//     PlcTask Outputs/GVL_iXlinker.Device_2_EtherCAT.Term_9_EK1100.Term_10_EK1122.Term_23_EK1100.Term_32_EL2258.MTO_Outputs_10x_Channel_6.Output_event_time[1] <-> MTO Outputs 10x Channel 6/Output event time 2
//     PlcTask Outputs/GVL_iXlinker.Device_2_EtherCAT.Term_9_EK1100.Term_10_EK1122.Term_23_EK1100.Term_32_EL2258.MTO_Outputs_10x_Channel_6.Output_event_time[2] <-> MTO Outputs 10x Channel 6/Output event time 3
//     PlcTask Outputs/GVL_iXlinker.Device_2_EtherCAT.Term_9_EK1100.Term_10_EK1122.Term_23_EK1100.Term_32_EL2258.MTO_Outputs_10x_Channel_6.Output_event_time[3] <-> MTO Outputs 10x Channel 6/Output event time 4
//     PlcTask Outputs/GVL_iXlinker.Device_2_EtherCAT.Term_9_EK1100.Term_10_EK1122.Term_23_EK1100.Term_32_EL2258.MTO_Outputs_10x_Channel_6.Output_event_time[4] <-> MTO Outputs 10x Channel 6/Output event time 5
//     PlcTask Outputs/GVL_iXlinker.Device_2_EtherCAT.Term_9_EK1100.Term_10_EK1122.Term_23_EK1100.Term_32_EL2258.MTO_Outputs_10x_Channel_6.Output_event_time[5] <-> MTO Outputs 10x Channel 6/Output event time 6
//     PlcTask Outputs/GVL_iXlinker.Device_2_EtherCAT.Term_9_EK1100.Term_10_EK1122.Term_23_EK1100.Term_32_EL2258.MTO_Outputs_10x_Channel_6.Output_event_time[6] <-> MTO Outputs 10x Channel 6/Output event time 7
//     PlcTask Outputs/GVL_iXlinker.Device_2_EtherCAT.Term_9_EK1100.Term_10_EK1122.Term_23_EK1100.Term_32_EL2258.MTO_Outputs_10x_Channel_6.Output_event_time[7] <-> MTO Outputs 10x Channel 6/Output event time 8
//     PlcTask Outputs/GVL_iXlinker.Device_2_EtherCAT.Term_9_EK1100.Term_10_EK1122.Term_23_EK1100.Term_32_EL2258.MTO_Outputs_10x_Channel_6.Output_event_time[8] <-> MTO Outputs 10x Channel 6/Output event time 9
//     PlcTask Outputs/GVL_iXlinker.Device_2_EtherCAT.Term_9_EK1100.Term_10_EK1122.Term_23_EK1100.Term_32_EL2258.MTO_Outputs_10x_Channel_6.Output_event_time[9] <-> MTO Outputs 10x Channel 6/Output event time 10
//     PlcTask Outputs/GVL_iXlinker.Device_2_EtherCAT.Term_9_EK1100.Term_10_EK1122.Term_23_EK1100.Term_32_EL2258.MTO_Outputs_10x_Channel_7.Output_event_time[0] <-> MTO Outputs 10x Channel 7/Output event time 1
//     PlcTask Outputs/GVL_iXlinker.Device_2_EtherCAT.Term_9_EK1100.Term_10_EK1122.Term_23_EK1100.Term_32_EL2258.MTO_Outputs_10x_Channel_7.Output_event_time[1] <-> MTO Outputs 10x Channel 7/Output event time 2
//     PlcTask Outputs/GVL_iXlinker.Device_2_EtherCAT.Term_9_EK1100.Term_10_EK1122.Term_23_EK1100.Term_32_EL2258.MTO_Outputs_10x_Channel_7.Output_event_time[2] <-> MTO Outputs 10x Channel 7/Output event time 3
//     PlcTask Outputs/GVL_iXlinker.Device_2_EtherCAT.Term_9_EK1100.Term_10_EK1122.Term_23_EK1100.Term_32_EL2258.MTO_Outputs_10x_Channel_7.Output_event_time[3] <-> MTO Outputs 10x Channel 7/Output event time 4
//     PlcTask Outputs/GVL_iXlinker.Device_2_EtherCAT.Term_9_EK1100.Term_10_EK1122.Term_23_EK1100.Term_32_EL2258.MTO_Outputs_10x_Channel_7.Output_event_time[4] <-> MTO Outputs 10x Channel 7/Output event time 5
//     PlcTask Outputs/GVL_iXlinker.Device_2_EtherCAT.Term_9_EK1100.Term_10_EK1122.Term_23_EK1100.Term_32_EL2258.MTO_Outputs_10x_Channel_7.Output_event_time[5] <-> MTO Outputs 10x Channel 7/Output event time 6
//     PlcTask Outputs/GVL_iXlinker.Device_2_EtherCAT.Term_9_EK1100.Term_10_EK1122.Term_23_EK1100.Term_32_EL2258.MTO_Outputs_10x_Channel_7.Output_event_time[6] <-> MTO Outputs 10x Channel 7/Output event time 7
//     PlcTask Outputs/GVL_iXlinker.Device_2_EtherCAT.Term_9_EK1100.Term_10_EK1122.Term_23_EK1100.Term_32_EL2258.MTO_Outputs_10x_Channel_7.Output_event_time[7] <-> MTO Outputs 10x Channel 7/Output event time 8
//     PlcTask Outputs/GVL_iXlinker.Device_2_EtherCAT.Term_9_EK1100.Term_10_EK1122.Term_23_EK1100.Term_32_EL2258.MTO_Outputs_10x_Channel_7.Output_event_time[8] <-> MTO Outputs 10x Channel 7/Output event time 9
//     PlcTask Outputs/GVL_iXlinker.Device_2_EtherCAT.Term_9_EK1100.Term_10_EK1122.Term_23_EK1100.Term_32_EL2258.MTO_Outputs_10x_Channel_7.Output_event_time[9] <-> MTO Outputs 10x Channel 7/Output event time 10
//     PlcTask Outputs/GVL_iXlinker.Device_2_EtherCAT.Term_9_EK1100.Term_10_EK1122.Term_23_EK1100.Term_32_EL2258.MTO_Outputs_10x_Channel_8.Output_event_time[0] <-> MTO Outputs 10x Channel 8/Output event time 1
//     PlcTask Outputs/GVL_iXlinker.Device_2_EtherCAT.Term_9_EK1100.Term_10_EK1122.Term_23_EK1100.Term_32_EL2258.MTO_Outputs_10x_Channel_8.Output_event_time[1] <-> MTO Outputs 10x Channel 8/Output event time 2
//     PlcTask Outputs/GVL_iXlinker.Device_2_EtherCAT.Term_9_EK1100.Term_10_EK1122.Term_23_EK1100.Term_32_EL2258.MTO_Outputs_10x_Channel_8.Output_event_time[2] <-> MTO Outputs 10x Channel 8/Output event time 3
//     PlcTask Outputs/GVL_iXlinker.Device_2_EtherCAT.Term_9_EK1100.Term_10_EK1122.Term_23_EK1100.Term_32_EL2258.MTO_Outputs_10x_Channel_8.Output_event_time[3] <-> MTO Outputs 10x Channel 8/Output event time 4
//     PlcTask Outputs/GVL_iXlinker.Device_2_EtherCAT.Term_9_EK1100.Term_10_EK1122.Term_23_EK1100.Term_32_EL2258.MTO_Outputs_10x_Channel_8.Output_event_time[4] <-> MTO Outputs 10x Channel 8/Output event time 5
//     PlcTask Outputs/GVL_iXlinker.Device_2_EtherCAT.Term_9_EK1100.Term_10_EK1122.Term_23_EK1100.Term_32_EL2258.MTO_Outputs_10x_Channel_8.Output_event_time[5] <-> MTO Outputs 10x Channel 8/Output event time 6
//     PlcTask Outputs/GVL_iXlinker.Device_2_EtherCAT.Term_9_EK1100.Term_10_EK1122.Term_23_EK1100.Term_32_EL2258.MTO_Outputs_10x_Channel_8.Output_event_time[6] <-> MTO Outputs 10x Channel 8/Output event time 7
//     PlcTask Outputs/GVL_iXlinker.Device_2_EtherCAT.Term_9_EK1100.Term_10_EK1122.Term_23_EK1100.Term_32_EL2258.MTO_Outputs_10x_Channel_8.Output_event_time[7] <-> MTO Outputs 10x Channel 8/Output event time 8
//     PlcTask Outputs/GVL_iXlinker.Device_2_EtherCAT.Term_9_EK1100.Term_10_EK1122.Term_23_EK1100.Term_32_EL2258.MTO_Outputs_10x_Channel_8.Output_event_time[8] <-> MTO Outputs 10x Channel 8/Output event time 9
//     PlcTask Outputs/GVL_iXlinker.Device_2_EtherCAT.Term_9_EK1100.Term_10_EK1122.Term_23_EK1100.Term_32_EL2258.MTO_Outputs_10x_Channel_8.Output_event_time[9] <-> MTO Outputs 10x Channel 8/Output event time 10
//     PlcTask Outputs/GVL_iXlinker.Device_2_EtherCAT.Term_9_EK1100.Term_10_EK1122.Term_23_EK1100.Term_32_EL2258.MTO_Outputs_10x_Channel_1.Outputs/Output_event_state_1 <-> MTO Outputs 10x Channel 1/Outputs/Output event state 1
//     PlcTask Outputs/GVL_iXlinker.Device_2_EtherCAT.Term_9_EK1100.Term_10_EK1122.Term_23_EK1100.Term_32_EL2258.MTO_Outputs_10x_Channel_1.Outputs/Output_event_state_10 <-> MTO Outputs 10x Channel 1/Outputs/Output event state 10
//     PlcTask Outputs/GVL_iXlinker.Device_2_EtherCAT.Term_9_EK1100.Term_10_EK1122.Term_23_EK1100.Term_32_EL2258.MTO_Outputs_10x_Channel_1.Outputs/Output_event_state_2 <-> MTO Outputs 10x Channel 1/Outputs/Output event state 2
//     PlcTask Outputs/GVL_iXlinker.Device_2_EtherCAT.Term_9_EK1100.Term_10_EK1122.Term_23_EK1100.Term_32_EL2258.MTO_Outputs_10x_Channel_1.Outputs/Output_event_state_3 <-> MTO Outputs 10x Channel 1/Outputs/Output event state 3
//     PlcTask Outputs/GVL_iXlinker.Device_2_EtherCAT.Term_9_EK1100.Term_10_EK1122.Term_23_EK1100.Term_32_EL2258.MTO_Outputs_10x_Channel_1.Outputs/Output_event_state_4 <-> MTO Outputs 10x Channel 1/Outputs/Output event state 4
//     PlcTask Outputs/GVL_iXlinker.Device_2_EtherCAT.Term_9_EK1100.Term_10_EK1122.Term_23_EK1100.Term_32_EL2258.MTO_Outputs_10x_Channel_1.Outputs/Output_event_state_5 <-> MTO Outputs 10x Channel 1/Outputs/Output event state 5
//     PlcTask Outputs/GVL_iXlinker.Device_2_EtherCAT.Term_9_EK1100.Term_10_EK1122.Term_23_EK1100.Term_32_EL2258.MTO_Outputs_10x_Channel_1.Outputs/Output_event_state_6 <-> MTO Outputs 10x Channel 1/Outputs/Output event state 6
//     PlcTask Outputs/GVL_iXlinker.Device_2_EtherCAT.Term_9_EK1100.Term_10_EK1122.Term_23_EK1100.Term_32_EL2258.MTO_Outputs_10x_Channel_1.Outputs/Output_event_state_7 <-> MTO Outputs 10x Channel 1/Outputs/Output event state 7
//     PlcTask Outputs/GVL_iXlinker.Device_2_EtherCAT.Term_9_EK1100.Term_10_EK1122.Term_23_EK1100.Term_32_EL2258.MTO_Outputs_10x_Channel_1.Outputs/Output_event_state_8 <-> MTO Outputs 10x Channel 1/Outputs/Output event state 8
//     PlcTask Outputs/GVL_iXlinker.Device_2_EtherCAT.Term_9_EK1100.Term_10_EK1122.Term_23_EK1100.Term_32_EL2258.MTO_Outputs_10x_Channel_1.Outputs/Output_event_state_9 <-> MTO Outputs 10x Channel 1/Outputs/Output event state 9
//     PlcTask Outputs/GVL_iXlinker.Device_2_EtherCAT.Term_9_EK1100.Term_10_EK1122.Term_23_EK1100.Term_32_EL2258.MTO_Outputs_10x_Channel_2.Outputs/Output_event_state_1 <-> MTO Outputs 10x Channel 2/Outputs/Output event state 1
//     PlcTask Outputs/GVL_iXlinker.Device_2_EtherCAT.Term_9_EK1100.Term_10_EK1122.Term_23_EK1100.Term_32_EL2258.MTO_Outputs_10x_Channel_2.Outputs/Output_event_state_10 <-> MTO Outputs 10x Channel 2/Outputs/Output event state 10
//     PlcTask Outputs/GVL_iXlinker.Device_2_EtherCAT.Term_9_EK1100.Term_10_EK1122.Term_23_EK1100.Term_32_EL2258.MTO_Outputs_10x_Channel_2.Outputs/Output_event_state_2 <-> MTO Outputs 10x Channel 2/Outputs/Output event state 2
//     PlcTask Outputs/GVL_iXlinker.Device_2_EtherCAT.Term_9_EK1100.Term_10_EK1122.Term_23_EK1100.Term_32_EL2258.MTO_Outputs_10x_Channel_2.Outputs/Output_event_state_3 <-> MTO Outputs 10x Channel 2/Outputs/Output event state 3
//     PlcTask Outputs/GVL_iXlinker.Device_2_EtherCAT.Term_9_EK1100.Term_10_EK1122.Term_23_EK1100.Term_32_EL2258.MTO_Outputs_10x_Channel_2.Outputs/Output_event_state_4 <-> MTO Outputs 10x Channel 2/Outputs/Output event state 4
//     PlcTask Outputs/GVL_iXlinker.Device_2_EtherCAT.Term_9_EK1100.Term_10_EK1122.Term_23_EK1100.Term_32_EL2258.MTO_Outputs_10x_Channel_2.Outputs/Output_event_state_5 <-> MTO Outputs 10x Channel 2/Outputs/Output event state 5
//     PlcTask Outputs/GVL_iXlinker.Device_2_EtherCAT.Term_9_EK1100.Term_10_EK1122.Term_23_EK1100.Term_32_EL2258.MTO_Outputs_10x_Channel_2.Outputs/Output_event_state_6 <-> MTO Outputs 10x Channel 2/Outputs/Output event state 6
//     PlcTask Outputs/GVL_iXlinker.Device_2_EtherCAT.Term_9_EK1100.Term_10_EK1122.Term_23_EK1100.Term_32_EL2258.MTO_Outputs_10x_Channel_2.Outputs/Output_event_state_7 <-> MTO Outputs 10x Channel 2/Outputs/Output event state 7
//     PlcTask Outputs/GVL_iXlinker.Device_2_EtherCAT.Term_9_EK1100.Term_10_EK1122.Term_23_EK1100.Term_32_EL2258.MTO_Outputs_10x_Channel_2.Outputs/Output_event_state_8 <-> MTO Outputs 10x Channel 2/Outputs/Output event state 8
//     PlcTask Outputs/GVL_iXlinker.Device_2_EtherCAT.Term_9_EK1100.Term_10_EK1122.Term_23_EK1100.Term_32_EL2258.MTO_Outputs_10x_Channel_2.Outputs/Output_event_state_9 <-> MTO Outputs 10x Channel 2/Outputs/Output event state 9
//     PlcTask Outputs/GVL_iXlinker.Device_2_EtherCAT.Term_9_EK1100.Term_10_EK1122.Term_23_EK1100.Term_32_EL2258.MTO_Outputs_10x_Channel_3.Outputs/Output_event_state_1 <-> MTO Outputs 10x Channel 3/Outputs/Output event state 1
//     PlcTask Outputs/GVL_iXlinker.Device_2_EtherCAT.Term_9_EK1100.Term_10_EK1122.Term_23_EK1100.Term_32_EL2258.MTO_Outputs_10x_Channel_3.Outputs/Output_event_state_10 <-> MTO Outputs 10x Channel 3/Outputs/Output event state 10
//     PlcTask Outputs/GVL_iXlinker.Device_2_EtherCAT.Term_9_EK1100.Term_10_EK1122.Term_23_EK1100.Term_32_EL2258.MTO_Outputs_10x_Channel_3.Outputs/Output_event_state_2 <-> MTO Outputs 10x Channel 3/Outputs/Output event state 2
//     PlcTask Outputs/GVL_iXlinker.Device_2_EtherCAT.Term_9_EK1100.Term_10_EK1122.Term_23_EK1100.Term_32_EL2258.MTO_Outputs_10x_Channel_3.Outputs/Output_event_state_3 <-> MTO Outputs 10x Channel 3/Outputs/Output event state 3
//     PlcTask Outputs/GVL_iXlinker.Device_2_EtherCAT.Term_9_EK1100.Term_10_EK1122.Term_23_EK1100.Term_32_EL2258.MTO_Outputs_10x_Channel_3.Outputs/Output_event_state_4 <-> MTO Outputs 10x Channel 3/Outputs/Output event state 4
//     PlcTask Outputs/GVL_iXlinker.Device_2_EtherCAT.Term_9_EK1100.Term_10_EK1122.Term_23_EK1100.Term_32_EL2258.MTO_Outputs_10x_Channel_3.Outputs/Output_event_state_5 <-> MTO Outputs 10x Channel 3/Outputs/Output event state 5
//     PlcTask Outputs/GVL_iXlinker.Device_2_EtherCAT.Term_9_EK1100.Term_10_EK1122.Term_23_EK1100.Term_32_EL2258.MTO_Outputs_10x_Channel_3.Outputs/Output_event_state_6 <-> MTO Outputs 10x Channel 3/Outputs/Output event state 6
//     PlcTask Outputs/GVL_iXlinker.Device_2_EtherCAT.Term_9_EK1100.Term_10_EK1122.Term_23_EK1100.Term_32_EL2258.MTO_Outputs_10x_Channel_3.Outputs/Output_event_state_7 <-> MTO Outputs 10x Channel 3/Outputs/Output event state 7
//     PlcTask Outputs/GVL_iXlinker.Device_2_EtherCAT.Term_9_EK1100.Term_10_EK1122.Term_23_EK1100.Term_32_EL2258.MTO_Outputs_10x_Channel_3.Outputs/Output_event_state_8 <-> MTO Outputs 10x Channel 3/Outputs/Output event state 8
//     PlcTask Outputs/GVL_iXlinker.Device_2_EtherCAT.Term_9_EK1100.Term_10_EK1122.Term_23_EK1100.Term_32_EL2258.MTO_Outputs_10x_Channel_3.Outputs/Output_event_state_9 <-> MTO Outputs 10x Channel 3/Outputs/Output event state 9
//     PlcTask Outputs/GVL_iXlinker.Device_2_EtherCAT.Term_9_EK1100.Term_10_EK1122.Term_23_EK1100.Term_32_EL2258.MTO_Outputs_10x_Channel_4.Outputs/Output_event_state_1 <-> MTO Outputs 10x Channel 4/Outputs/Output event state 1
//     PlcTask Outputs/GVL_iXlinker.Device_2_EtherCAT.Term_9_EK1100.Term_10_EK1122.Term_23_EK1100.Term_32_EL2258.MTO_Outputs_10x_Channel_4.Outputs/Output_event_state_10 <-> MTO Outputs 10x Channel 4/Outputs/Output event state 10
//     PlcTask Outputs/GVL_iXlinker.Device_2_EtherCAT.Term_9_EK1100.Term_10_EK1122.Term_23_EK1100.Term_32_EL2258.MTO_Outputs_10x_Channel_4.Outputs/Output_event_state_2 <-> MTO Outputs 10x Channel 4/Outputs/Output event state 2
//     PlcTask Outputs/GVL_iXlinker.Device_2_EtherCAT.Term_9_EK1100.Term_10_EK1122.Term_23_EK1100.Term_32_EL2258.MTO_Outputs_10x_Channel_4.Outputs/Output_event_state_3 <-> MTO Outputs 10x Channel 4/Outputs/Output event state 3
//     PlcTask Outputs/GVL_iXlinker.Device_2_EtherCAT.Term_9_EK1100.Term_10_EK1122.Term_23_EK1100.Term_32_EL2258.MTO_Outputs_10x_Channel_4.Outputs/Output_event_state_4 <-> MTO Outputs 10x Channel 4/Outputs/Output event state 4
//     PlcTask Outputs/GVL_iXlinker.Device_2_EtherCAT.Term_9_EK1100.Term_10_EK1122.Term_23_EK1100.Term_32_EL2258.MTO_Outputs_10x_Channel_4.Outputs/Output_event_state_5 <-> MTO Outputs 10x Channel 4/Outputs/Output event state 5
//     PlcTask Outputs/GVL_iXlinker.Device_2_EtherCAT.Term_9_EK1100.Term_10_EK1122.Term_23_EK1100.Term_32_EL2258.MTO_Outputs_10x_Channel_4.Outputs/Output_event_state_6 <-> MTO Outputs 10x Channel 4/Outputs/Output event state 6
//     PlcTask Outputs/GVL_iXlinker.Device_2_EtherCAT.Term_9_EK1100.Term_10_EK1122.Term_23_EK1100.Term_32_EL2258.MTO_Outputs_10x_Channel_4.Outputs/Output_event_state_7 <-> MTO Outputs 10x Channel 4/Outputs/Output event state 7
//     PlcTask Outputs/GVL_iXlinker.Device_2_EtherCAT.Term_9_EK1100.Term_10_EK1122.Term_23_EK1100.Term_32_EL2258.MTO_Outputs_10x_Channel_4.Outputs/Output_event_state_8 <-> MTO Outputs 10x Channel 4/Outputs/Output event state 8
//     PlcTask Outputs/GVL_iXlinker.Device_2_EtherCAT.Term_9_EK1100.Term_10_EK1122.Term_23_EK1100.Term_32_EL2258.MTO_Outputs_10x_Channel_4.Outputs/Output_event_state_9 <-> MTO Outputs 10x Channel 4/Outputs/Output event state 9
//     PlcTask Outputs/GVL_iXlinker.Device_2_EtherCAT.Term_9_EK1100.Term_10_EK1122.Term_23_EK1100.Term_32_EL2258.MTO_Outputs_10x_Channel_5.Outputs/Output_event_state_1 <-> MTO Outputs 10x Channel 5/Outputs/Output event state 1
//     PlcTask Outputs/GVL_iXlinker.Device_2_EtherCAT.Term_9_EK1100.Term_10_EK1122.Term_23_EK1100.Term_32_EL2258.MTO_Outputs_10x_Channel_5.Outputs/Output_event_state_10 <-> MTO Outputs 10x Channel 5/Outputs/Output event state 10
//     PlcTask Outputs/GVL_iXlinker.Device_2_EtherCAT.Term_9_EK1100.Term_10_EK1122.Term_23_EK1100.Term_32_EL2258.MTO_Outputs_10x_Channel_5.Outputs/Output_event_state_2 <-> MTO Outputs 10x Channel 5/Outputs/Output event state 2
//     PlcTask Outputs/GVL_iXlinker.Device_2_EtherCAT.Term_9_EK1100.Term_10_EK1122.Term_23_EK1100.Term_32_EL2258.MTO_Outputs_10x_Channel_5.Outputs/Output_event_state_3 <-> MTO Outputs 10x Channel 5/Outputs/Output event state 3
//     PlcTask Outputs/GVL_iXlinker.Device_2_EtherCAT.Term_9_EK1100.Term_10_EK1122.Term_23_EK1100.Term_32_EL2258.MTO_Outputs_10x_Channel_5.Outputs/Output_event_state_4 <-> MTO Outputs 10x Channel 5/Outputs/Output event state 4
//     PlcTask Outputs/GVL_iXlinker.Device_2_EtherCAT.Term_9_EK1100.Term_10_EK1122.Term_23_EK1100.Term_32_EL2258.MTO_Outputs_10x_Channel_5.Outputs/Output_event_state_5 <-> MTO Outputs 10x Channel 5/Outputs/Output event state 5
//     PlcTask Outputs/GVL_iXlinker.Device_2_EtherCAT.Term_9_EK1100.Term_10_EK1122.Term_23_EK1100.Term_32_EL2258.MTO_Outputs_10x_Channel_5.Outputs/Output_event_state_6 <-> MTO Outputs 10x Channel 5/Outputs/Output event state 6
//     PlcTask Outputs/GVL_iXlinker.Device_2_EtherCAT.Term_9_EK1100.Term_10_EK1122.Term_23_EK1100.Term_32_EL2258.MTO_Outputs_10x_Channel_5.Outputs/Output_event_state_7 <-> MTO Outputs 10x Channel 5/Outputs/Output event state 7
//     PlcTask Outputs/GVL_iXlinker.Device_2_EtherCAT.Term_9_EK1100.Term_10_EK1122.Term_23_EK1100.Term_32_EL2258.MTO_Outputs_10x_Channel_5.Outputs/Output_event_state_8 <-> MTO Outputs 10x Channel 5/Outputs/Output event state 8
//     PlcTask Outputs/GVL_iXlinker.Device_2_EtherCAT.Term_9_EK1100.Term_10_EK1122.Term_23_EK1100.Term_32_EL2258.MTO_Outputs_10x_Channel_5.Outputs/Output_event_state_9 <-> MTO Outputs 10x Channel 5/Outputs/Output event state 9
//     PlcTask Outputs/GVL_iXlinker.Device_2_EtherCAT.Term_9_EK1100.Term_10_EK1122.Term_23_EK1100.Term_32_EL2258.MTO_Outputs_10x_Channel_6.Outputs/Output_event_state_1 <-> MTO Outputs 10x Channel 6/Outputs/Output event state 1
//     PlcTask Outputs/GVL_iXlinker.Device_2_EtherCAT.Term_9_EK1100.Term_10_EK1122.Term_23_EK1100.Term_32_EL2258.MTO_Outputs_10x_Channel_6.Outputs/Output_event_state_10 <-> MTO Outputs 10x Channel 6/Outputs/Output event state 10
//     PlcTask Outputs/GVL_iXlinker.Device_2_EtherCAT.Term_9_EK1100.Term_10_EK1122.Term_23_EK1100.Term_32_EL2258.MTO_Outputs_10x_Channel_6.Outputs/Output_event_state_2 <-> MTO Outputs 10x Channel 6/Outputs/Output event state 2
//     PlcTask Outputs/GVL_iXlinker.Device_2_EtherCAT.Term_9_EK1100.Term_10_EK1122.Term_23_EK1100.Term_32_EL2258.MTO_Outputs_10x_Channel_6.Outputs/Output_event_state_3 <-> MTO Outputs 10x Channel 6/Outputs/Output event state 3
//     PlcTask Outputs/GVL_iXlinker.Device_2_EtherCAT.Term_9_EK1100.Term_10_EK1122.Term_23_EK1100.Term_32_EL2258.MTO_Outputs_10x_Channel_6.Outputs/Output_event_state_4 <-> MTO Outputs 10x Channel 6/Outputs/Output event state 4
//     PlcTask Outputs/GVL_iXlinker.Device_2_EtherCAT.Term_9_EK1100.Term_10_EK1122.Term_23_EK1100.Term_32_EL2258.MTO_Outputs_10x_Channel_6.Outputs/Output_event_state_5 <-> MTO Outputs 10x Channel 6/Outputs/Output event state 5
//     PlcTask Outputs/GVL_iXlinker.Device_2_EtherCAT.Term_9_EK1100.Term_10_EK1122.Term_23_EK1100.Term_32_EL2258.MTO_Outputs_10x_Channel_6.Outputs/Output_event_state_6 <-> MTO Outputs 10x Channel 6/Outputs/Output event state 6
//     PlcTask Outputs/GVL_iXlinker.Device_2_EtherCAT.Term_9_EK1100.Term_10_EK1122.Term_23_EK1100.Term_32_EL2258.MTO_Outputs_10x_Channel_6.Outputs/Output_event_state_7 <-> MTO Outputs 10x Channel 6/Outputs/Output event state 7
//     PlcTask Outputs/GVL_iXlinker.Device_2_EtherCAT.Term_9_EK1100.Term_10_EK1122.Term_23_EK1100.Term_32_EL2258.MTO_Outputs_10x_Channel_6.Outputs/Output_event_state_8 <-> MTO Outputs 10x Channel 6/Outputs/Output event state 8
//     PlcTask Outputs/GVL_iXlinker.Device_2_EtherCAT.Term_9_EK1100.Term_10_EK1122.Term_23_EK1100.Term_32_EL2258.MTO_Outputs_10x_Channel_6.Outputs/Output_event_state_9 <-> MTO Outputs 10x Channel 6/Outputs/Output event state 9
//     PlcTask Outputs/GVL_iXlinker.Device_2_EtherCAT.Term_9_EK1100.Term_10_EK1122.Term_23_EK1100.Term_32_EL2258.MTO_Outputs_10x_Channel_7.Outputs/Output_event_state_1 <-> MTO Outputs 10x Channel 7/Outputs/Output event state 1
//     PlcTask Outputs/GVL_iXlinker.Device_2_EtherCAT.Term_9_EK1100.Term_10_EK1122.Term_23_EK1100.Term_32_EL2258.MTO_Outputs_10x_Channel_7.Outputs/Output_event_state_10 <-> MTO Outputs 10x Channel 7/Outputs/Output event state 10
//     PlcTask Outputs/GVL_iXlinker.Device_2_EtherCAT.Term_9_EK1100.Term_10_EK1122.Term_23_EK1100.Term_32_EL2258.MTO_Outputs_10x_Channel_7.Outputs/Output_event_state_2 <-> MTO Outputs 10x Channel 7/Outputs/Output event state 2
//     PlcTask Outputs/GVL_iXlinker.Device_2_EtherCAT.Term_9_EK1100.Term_10_EK1122.Term_23_EK1100.Term_32_EL2258.MTO_Outputs_10x_Channel_7.Outputs/Output_event_state_3 <-> MTO Outputs 10x Channel 7/Outputs/Output event state 3
//     PlcTask Outputs/GVL_iXlinker.Device_2_EtherCAT.Term_9_EK1100.Term_10_EK1122.Term_23_EK1100.Term_32_EL2258.MTO_Outputs_10x_Channel_7.Outputs/Output_event_state_4 <-> MTO Outputs 10x Channel 7/Outputs/Output event state 4
//     PlcTask Outputs/GVL_iXlinker.Device_2_EtherCAT.Term_9_EK1100.Term_10_EK1122.Term_23_EK1100.Term_32_EL2258.MTO_Outputs_10x_Channel_7.Outputs/Output_event_state_5 <-> MTO Outputs 10x Channel 7/Outputs/Output event state 5
//     PlcTask Outputs/GVL_iXlinker.Device_2_EtherCAT.Term_9_EK1100.Term_10_EK1122.Term_23_EK1100.Term_32_EL2258.MTO_Outputs_10x_Channel_7.Outputs/Output_event_state_6 <-> MTO Outputs 10x Channel 7/Outputs/Output event state 6
//     PlcTask Outputs/GVL_iXlinker.Device_2_EtherCAT.Term_9_EK1100.Term_10_EK1122.Term_23_EK1100.Term_32_EL2258.MTO_Outputs_10x_Channel_7.Outputs/Output_event_state_7 <-> MTO Outputs 10x Channel 7/Outputs/Output event state 7
//     PlcTask Outputs/GVL_iXlinker.Device_2_EtherCAT.Term_9_EK1100.Term_10_EK1122.Term_23_EK1100.Term_32_EL2258.MTO_Outputs_10x_Channel_7.Outputs/Output_event_state_8 <-> MTO Outputs 10x Channel 7/Outputs/Output event state 8
//     PlcTask Outputs/GVL_iXlinker.Device_2_EtherCAT.Term_9_EK1100.Term_10_EK1122.Term_23_EK1100.Term_32_EL2258.MTO_Outputs_10x_Channel_7.Outputs/Output_event_state_9 <-> MTO Outputs 10x Channel 7/Outputs/Output event state 9
//     PlcTask Outputs/GVL_iXlinker.Device_2_EtherCAT.Term_9_EK1100.Term_10_EK1122.Term_23_EK1100.Term_32_EL2258.MTO_Outputs_10x_Channel_8.Outputs/Output_event_state_1 <-> MTO Outputs 10x Channel 8/Outputs/Output event state 1
//     PlcTask Outputs/GVL_iXlinker.Device_2_EtherCAT.Term_9_EK1100.Term_10_EK1122.Term_23_EK1100.Term_32_EL2258.MTO_Outputs_10x_Channel_8.Outputs/Output_event_state_10 <-> MTO Outputs 10x Channel 8/Outputs/Output event state 10
//     PlcTask Outputs/GVL_iXlinker.Device_2_EtherCAT.Term_9_EK1100.Term_10_EK1122.Term_23_EK1100.Term_32_EL2258.MTO_Outputs_10x_Channel_8.Outputs/Output_event_state_2 <-> MTO Outputs 10x Channel 8/Outputs/Output event state 2
//     PlcTask Outputs/GVL_iXlinker.Device_2_EtherCAT.Term_9_EK1100.Term_10_EK1122.Term_23_EK1100.Term_32_EL2258.MTO_Outputs_10x_Channel_8.Outputs/Output_event_state_3 <-> MTO Outputs 10x Channel 8/Outputs/Output event state 3
//     PlcTask Outputs/GVL_iXlinker.Device_2_EtherCAT.Term_9_EK1100.Term_10_EK1122.Term_23_EK1100.Term_32_EL2258.MTO_Outputs_10x_Channel_8.Outputs/Output_event_state_4 <-> MTO Outputs 10x Channel 8/Outputs/Output event state 4
//     PlcTask Outputs/GVL_iXlinker.Device_2_EtherCAT.Term_9_EK1100.Term_10_EK1122.Term_23_EK1100.Term_32_EL2258.MTO_Outputs_10x_Channel_8.Outputs/Output_event_state_5 <-> MTO Outputs 10x Channel 8/Outputs/Output event state 5
//     PlcTask Outputs/GVL_iXlinker.Device_2_EtherCAT.Term_9_EK1100.Term_10_EK1122.Term_23_EK1100.Term_32_EL2258.MTO_Outputs_10x_Channel_8.Outputs/Output_event_state_6 <-> MTO Outputs 10x Channel 8/Outputs/Output event state 6
//     PlcTask Outputs/GVL_iXlinker.Device_2_EtherCAT.Term_9_EK1100.Term_10_EK1122.Term_23_EK1100.Term_32_EL2258.MTO_Outputs_10x_Channel_8.Outputs/Output_event_state_7 <-> MTO Outputs 10x Channel 8/Outputs/Output event state 7
//     PlcTask Outputs/GVL_iXlinker.Device_2_EtherCAT.Term_9_EK1100.Term_10_EK1122.Term_23_EK1100.Term_32_EL2258.MTO_Outputs_10x_Channel_8.Outputs/Output_event_state_8 <-> MTO Outputs 10x Channel 8/Outputs/Output event state 8
//     PlcTask Outputs/GVL_iXlinker.Device_2_EtherCAT.Term_9_EK1100.Term_10_EK1122.Term_23_EK1100.Term_32_EL2258.MTO_Outputs_10x_Channel_8.Outputs/Output_event_state_9 <-> MTO Outputs 10x Channel 8/Outputs/Output event state 9
//   Plc1/Plc1 Instance <-> Device 2 (EtherCAT)/Term 9 (EK1100)/Term 10 (EK1122)/Term 23 (EK1100)/Term 33 (EL3164)
//     PlcTask Inputs/GVL_iXlinker.Device_2_EtherCAT.Term_9_EK1100.Term_10_EK1122.Term_23_EK1100.Term_33_EL3164.AI_Standard_Channel_{1..4}.Status/Error <-> AI Standard Channel {1..4}/Status/Error  (4 links)
//     PlcTask Inputs/GVL_iXlinker.Device_2_EtherCAT.Term_9_EK1100.Term_10_EK1122.Term_23_EK1100.Term_33_EL3164.AI_Standard_Channel_1.Status/Limit_1 <-> AI Standard Channel 1/Status/Limit 1
//     PlcTask Inputs/GVL_iXlinker.Device_2_EtherCAT.Term_9_EK1100.Term_10_EK1122.Term_23_EK1100.Term_33_EL3164.AI_Standard_Channel_1.Status/Limit_2 <-> AI Standard Channel 1/Status/Limit 2
//     PlcTask Inputs/GVL_iXlinker.Device_2_EtherCAT.Term_9_EK1100.Term_10_EK1122.Term_23_EK1100.Term_33_EL3164.AI_Standard_Channel_2.Status/Limit_1 <-> AI Standard Channel 2/Status/Limit 1
//     PlcTask Inputs/GVL_iXlinker.Device_2_EtherCAT.Term_9_EK1100.Term_10_EK1122.Term_23_EK1100.Term_33_EL3164.AI_Standard_Channel_2.Status/Limit_2 <-> AI Standard Channel 2/Status/Limit 2
//     PlcTask Inputs/GVL_iXlinker.Device_2_EtherCAT.Term_9_EK1100.Term_10_EK1122.Term_23_EK1100.Term_33_EL3164.AI_Standard_Channel_3.Status/Limit_1 <-> AI Standard Channel 3/Status/Limit 1
//     PlcTask Inputs/GVL_iXlinker.Device_2_EtherCAT.Term_9_EK1100.Term_10_EK1122.Term_23_EK1100.Term_33_EL3164.AI_Standard_Channel_3.Status/Limit_2 <-> AI Standard Channel 3/Status/Limit 2
//     PlcTask Inputs/GVL_iXlinker.Device_2_EtherCAT.Term_9_EK1100.Term_10_EK1122.Term_23_EK1100.Term_33_EL3164.AI_Standard_Channel_4.Status/Limit_1 <-> AI Standard Channel 4/Status/Limit 1
//     PlcTask Inputs/GVL_iXlinker.Device_2_EtherCAT.Term_9_EK1100.Term_10_EK1122.Term_23_EK1100.Term_33_EL3164.AI_Standard_Channel_4.Status/Limit_2 <-> AI Standard Channel 4/Status/Limit 2
//     PlcTask Inputs/GVL_iXlinker.Device_2_EtherCAT.Term_9_EK1100.Term_10_EK1122.Term_23_EK1100.Term_33_EL3164.AI_Standard_Channel_{1..4}.Status/Overrange <-> AI Standard Channel {1..4}/Status/Overrange  (4 links)
//     PlcTask Inputs/GVL_iXlinker.Device_2_EtherCAT.Term_9_EK1100.Term_10_EK1122.Term_23_EK1100.Term_33_EL3164.AI_Standard_Channel_{1..4}.Status/Sync_error <-> AI Standard Channel {1..4}/Status/Sync error  (4 links)
//     PlcTask Inputs/GVL_iXlinker.Device_2_EtherCAT.Term_9_EK1100.Term_10_EK1122.Term_23_EK1100.Term_33_EL3164.AI_Standard_Channel_{1..4}.Status/TxPDO_State <-> AI Standard Channel {1..4}/Status/TxPDO State  (4 links)
//     PlcTask Inputs/GVL_iXlinker.Device_2_EtherCAT.Term_9_EK1100.Term_10_EK1122.Term_23_EK1100.Term_33_EL3164.AI_Standard_Channel_{1..4}.Status/TxPDO_Toggle <-> AI Standard Channel {1..4}/Status/TxPDO Toggle  (4 links)
//     PlcTask Inputs/GVL_iXlinker.Device_2_EtherCAT.Term_9_EK1100.Term_10_EK1122.Term_23_EK1100.Term_33_EL3164.AI_Standard_Channel_{1..4}.Status/Underrange <-> AI Standard Channel {1..4}/Status/Underrange  (4 links)
//     PlcTask Inputs/GVL_iXlinker.Device_2_EtherCAT.Term_9_EK1100.Term_10_EK1122.Term_23_EK1100.Term_33_EL3164.AI_Standard_Channel_{1..4}.Value <-> AI Standard Channel {1..4}/Value  (4 links)
//     PlcTask Inputs/GVL_iXlinker.Device_2_EtherCAT.Term_9_EK1100.Term_10_EK1122.Term_23_EK1100.Term_33_EL3164.InfoData.AdsAddr <-> InfoData/AdsAddr
//     PlcTask Inputs/GVL_iXlinker.Device_2_EtherCAT.Term_9_EK1100.Term_10_EK1122.Term_23_EK1100.Term_33_EL3164.InfoData.State <-> InfoData/State
//     PlcTask Inputs/GVL_iXlinker.Device_2_EtherCAT.Term_9_EK1100.Term_10_EK1122.Term_23_EK1100.Term_33_EL3164.WcState.InputToggle <-> WcState/InputToggle
//     PlcTask Inputs/GVL_iXlinker.Device_2_EtherCAT.Term_9_EK1100.Term_10_EK1122.Term_23_EK1100.Term_33_EL3164.WcState.WcState <-> WcState/WcState
//   Plc1/Plc1 Instance <-> Device 2 (EtherCAT)/Term 9 (EK1100)/Term 10 (EK1122)/Term 23 (EK1100)/Term 40 (EK1110)
//     PlcTask Inputs/GVL_iXlinker.Device_2_EtherCAT.Term_9_EK1100.Term_10_EK1122.Term_23_EK1100.Term_40_EK1110.InfoData.State <-> InfoData/State
//   Plc1/Plc1 Instance <-> Device 2 (EtherCAT)/Term 9 (EK1100)/Term 10 (EK1122)/Term 42 (EK1100)
//     PlcTask Inputs/GVL_iXlinker.Device_2_EtherCAT.Term_9_EK1100.Term_10_EK1122.Term_42_EK1100.InfoData.State <-> InfoData/State
//   Plc1/Plc1 Instance <-> Device 2 (EtherCAT)/Term 9 (EK1100)/Term 10 (EK1122)/Term 42 (EK1100)/Term 43 (EL1008)
//     PlcTask Inputs/GVL_iXlinker.Device_2_EtherCAT.Term_9_EK1100.Term_10_EK1122.Term_42_EK1100.Term_43_EL1008.Channel_{1..8}.Input <-> Channel {1..8}/Input  (8 links)
//     PlcTask Inputs/GVL_iXlinker.Device_2_EtherCAT.Term_9_EK1100.Term_10_EK1122.Term_42_EK1100.Term_43_EL1008.InfoData.State <-> InfoData/State
//     PlcTask Inputs/GVL_iXlinker.Device_2_EtherCAT.Term_9_EK1100.Term_10_EK1122.Term_42_EK1100.Term_43_EL1008.WcState.InputToggle <-> WcState/InputToggle
//     PlcTask Inputs/GVL_iXlinker.Device_2_EtherCAT.Term_9_EK1100.Term_10_EK1122.Term_42_EK1100.Term_43_EL1008.WcState.WcState <-> WcState/WcState
//   Plc1/Plc1 Instance <-> Device 2 (EtherCAT)/Term 9 (EK1100)/Term 10 (EK1122)/Term 42 (EK1100)/Term 44 (EL1008)
//     PlcTask Inputs/GVL_iXlinker.Device_2_EtherCAT.Term_9_EK1100.Term_10_EK1122.Term_42_EK1100.Term_44_EL1008.Channel_{1..8}.Input <-> Channel {1..8}/Input  (8 links)
//     PlcTask Inputs/GVL_iXlinker.Device_2_EtherCAT.Term_9_EK1100.Term_10_EK1122.Term_42_EK1100.Term_44_EL1008.InfoData.State <-> InfoData/State
//     PlcTask Inputs/GVL_iXlinker.Device_2_EtherCAT.Term_9_EK1100.Term_10_EK1122.Term_42_EK1100.Term_44_EL1008.WcState.InputToggle <-> WcState/InputToggle
//     PlcTask Inputs/GVL_iXlinker.Device_2_EtherCAT.Term_9_EK1100.Term_10_EK1122.Term_42_EK1100.Term_44_EL1008.WcState.WcState <-> WcState/WcState
//   Plc1/Plc1 Instance <-> Device 2 (EtherCAT)/Term 9 (EK1100)/Term 34 (EL3403)
//     PlcTask Inputs/GVL_iXlinker.Device_2_EtherCAT.Term_9_EK1100.Term_34_EL3403.InfoData.AdsAddr <-> InfoData/AdsAddr
//     PlcTask Inputs/GVL_iXlinker.Device_2_EtherCAT.Term_9_EK1100.Term_34_EL3403.InfoData.State <-> InfoData/State
//     PlcTask Inputs/GVL_iXlinker.Device_2_EtherCAT.Term_9_EK1100.Term_34_EL3403.PM_Inputs_Channel_1.Active_power <-> PM Inputs Channel 1/Active power
//     PlcTask Inputs/GVL_iXlinker.Device_2_EtherCAT.Term_9_EK1100.Term_34_EL3403.PM_Inputs_Channel_2.Active_power <-> PM Inputs Channel 2/Active power
//     PlcTask Inputs/GVL_iXlinker.Device_2_EtherCAT.Term_9_EK1100.Term_34_EL3403.PM_Inputs_Channel_3.Active_power <-> PM Inputs Channel 3/Active power
//     PlcTask Inputs/GVL_iXlinker.Device_2_EtherCAT.Term_9_EK1100.Term_34_EL3403.PM_Inputs_Channel_1.Current <-> PM Inputs Channel 1/Current
//     PlcTask Inputs/GVL_iXlinker.Device_2_EtherCAT.Term_9_EK1100.Term_34_EL3403.PM_Inputs_Channel_2.Current <-> PM Inputs Channel 2/Current
//     PlcTask Inputs/GVL_iXlinker.Device_2_EtherCAT.Term_9_EK1100.Term_34_EL3403.PM_Inputs_Channel_3.Current <-> PM Inputs Channel 3/Current
//     PlcTask Inputs/GVL_iXlinker.Device_2_EtherCAT.Term_9_EK1100.Term_34_EL3403.PM_Inputs_Channel_1.Index <-> PM Inputs Channel 1/Index
//     PlcTask Inputs/GVL_iXlinker.Device_2_EtherCAT.Term_9_EK1100.Term_34_EL3403.PM_Inputs_Channel_2.Index <-> PM Inputs Channel 2/Index
//     PlcTask Inputs/GVL_iXlinker.Device_2_EtherCAT.Term_9_EK1100.Term_34_EL3403.PM_Inputs_Channel_3.Index <-> PM Inputs Channel 3/Index
//     PlcTask Inputs/GVL_iXlinker.Device_2_EtherCAT.Term_9_EK1100.Term_34_EL3403.PM_Inputs_Channel_1.TxPDO_Toggle <-> PM Inputs Channel 1/TxPDO Toggle
//     PlcTask Inputs/GVL_iXlinker.Device_2_EtherCAT.Term_9_EK1100.Term_34_EL3403.PM_Inputs_Channel_2.TxPDO_Toggle <-> PM Inputs Channel 2/TxPDO Toggle
//     PlcTask Inputs/GVL_iXlinker.Device_2_EtherCAT.Term_9_EK1100.Term_34_EL3403.PM_Inputs_Channel_3.TxPDO_Toggle <-> PM Inputs Channel 3/TxPDO Toggle
//     PlcTask Inputs/GVL_iXlinker.Device_2_EtherCAT.Term_9_EK1100.Term_34_EL3403.PM_Inputs_Channel_1.Variant_value <-> PM Inputs Channel 1/Variant value
//     PlcTask Inputs/GVL_iXlinker.Device_2_EtherCAT.Term_9_EK1100.Term_34_EL3403.PM_Inputs_Channel_2.Variant_value <-> PM Inputs Channel 2/Variant value
//     PlcTask Inputs/GVL_iXlinker.Device_2_EtherCAT.Term_9_EK1100.Term_34_EL3403.PM_Inputs_Channel_3.Variant_value <-> PM Inputs Channel 3/Variant value
//     PlcTask Inputs/GVL_iXlinker.Device_2_EtherCAT.Term_9_EK1100.Term_34_EL3403.PM_Inputs_Channel_1.Voltage <-> PM Inputs Channel 1/Voltage
//     PlcTask Inputs/GVL_iXlinker.Device_2_EtherCAT.Term_9_EK1100.Term_34_EL3403.PM_Inputs_Channel_2.Voltage <-> PM Inputs Channel 2/Voltage
//     PlcTask Inputs/GVL_iXlinker.Device_2_EtherCAT.Term_9_EK1100.Term_34_EL3403.PM_Inputs_Channel_3.Voltage <-> PM Inputs Channel 3/Voltage
//     PlcTask Inputs/GVL_iXlinker.Device_2_EtherCAT.Term_9_EK1100.Term_34_EL3403.PM_Status_data.Missing_zero_crossing_A <-> PM Status data/Missing zero crossing A
//     PlcTask Inputs/GVL_iXlinker.Device_2_EtherCAT.Term_9_EK1100.Term_34_EL3403.PM_Status_data.Missing_zero_crossing_B <-> PM Status data/Missing zero crossing B
//     PlcTask Inputs/GVL_iXlinker.Device_2_EtherCAT.Term_9_EK1100.Term_34_EL3403.PM_Status_data.Missing_zero_crossing_C <-> PM Status data/Missing zero crossing C
//     PlcTask Inputs/GVL_iXlinker.Device_2_EtherCAT.Term_9_EK1100.Term_34_EL3403.PM_Status_data.Phase_sequence_error <-> PM Status data/Phase sequence error
//     PlcTask Inputs/GVL_iXlinker.Device_2_EtherCAT.Term_9_EK1100.Term_34_EL3403.WcState.InputToggle <-> WcState/InputToggle
//     PlcTask Inputs/GVL_iXlinker.Device_2_EtherCAT.Term_9_EK1100.Term_34_EL3403.WcState.WcState <-> WcState/WcState
//     PlcTask Outputs/GVL_iXlinker.Device_2_EtherCAT.Term_9_EK1100.Term_34_EL3403.PM_Outputs_Channel_1.Index <-> PM Outputs Channel 1/Index
//     PlcTask Outputs/GVL_iXlinker.Device_2_EtherCAT.Term_9_EK1100.Term_34_EL3403.PM_Outputs_Channel_2.Index <-> PM Outputs Channel 2/Index
//     PlcTask Outputs/GVL_iXlinker.Device_2_EtherCAT.Term_9_EK1100.Term_34_EL3403.PM_Outputs_Channel_3.Index <-> PM Outputs Channel 3/Index
//   Plc1/Plc1 Instance <-> Device 2 (EtherCAT)/Term 9 (EK1100)/Term 35 (EL6001)
//     PlcTask Inputs/GVL_iXlinker.Device_2_EtherCAT.Term_9_EK1100.Term_35_EL6001.COM_Inputs.Data_In[{0..21}] <-> COM Inputs/Data In {0..21}  (22 links)
//     PlcTask Inputs/GVL_iXlinker.Device_2_EtherCAT.Term_9_EK1100.Term_35_EL6001.COM_Inputs.Status/Buffer_full <-> COM Inputs/Status/Buffer full
//     PlcTask Inputs/GVL_iXlinker.Device_2_EtherCAT.Term_9_EK1100.Term_35_EL6001.COM_Inputs.Status/Framing_error <-> COM Inputs/Status/Framing error
//     PlcTask Inputs/GVL_iXlinker.Device_2_EtherCAT.Term_9_EK1100.Term_35_EL6001.COM_Inputs.Status/Init_accepted <-> COM Inputs/Status/Init accepted
//     PlcTask Inputs/GVL_iXlinker.Device_2_EtherCAT.Term_9_EK1100.Term_35_EL6001.COM_Inputs.Status/Input_length <-> COM Inputs/Status/Input length
//     PlcTask Inputs/GVL_iXlinker.Device_2_EtherCAT.Term_9_EK1100.Term_35_EL6001.COM_Inputs.Status/Overrun_error <-> COM Inputs/Status/Overrun error
//     PlcTask Inputs/GVL_iXlinker.Device_2_EtherCAT.Term_9_EK1100.Term_35_EL6001.COM_Inputs.Status/Parity_error <-> COM Inputs/Status/Parity error
//     PlcTask Inputs/GVL_iXlinker.Device_2_EtherCAT.Term_9_EK1100.Term_35_EL6001.COM_Inputs.Status/Receive_request <-> COM Inputs/Status/Receive request
//     PlcTask Inputs/GVL_iXlinker.Device_2_EtherCAT.Term_9_EK1100.Term_35_EL6001.COM_Inputs.Status/Transmit_accepted <-> COM Inputs/Status/Transmit accepted
//     PlcTask Inputs/GVL_iXlinker.Device_2_EtherCAT.Term_9_EK1100.Term_35_EL6001.InfoData.AdsAddr <-> InfoData/AdsAddr
//     PlcTask Inputs/GVL_iXlinker.Device_2_EtherCAT.Term_9_EK1100.Term_35_EL6001.InfoData.State <-> InfoData/State
//     PlcTask Inputs/GVL_iXlinker.Device_2_EtherCAT.Term_9_EK1100.Term_35_EL6001.WcState.InputToggle <-> WcState/InputToggle
//     PlcTask Inputs/GVL_iXlinker.Device_2_EtherCAT.Term_9_EK1100.Term_35_EL6001.WcState.WcState <-> WcState/WcState
//     PlcTask Outputs/GVL_iXlinker.Device_2_EtherCAT.Term_9_EK1100.Term_35_EL6001.COM_Outputs.Ctrl/Init_request <-> COM Outputs/Ctrl/Init request
//     PlcTask Outputs/GVL_iXlinker.Device_2_EtherCAT.Term_9_EK1100.Term_35_EL6001.COM_Outputs.Ctrl/Output_length <-> COM Outputs/Ctrl/Output length
//     PlcTask Outputs/GVL_iXlinker.Device_2_EtherCAT.Term_9_EK1100.Term_35_EL6001.COM_Outputs.Ctrl/Receive_accepted <-> COM Outputs/Ctrl/Receive accepted
//     PlcTask Outputs/GVL_iXlinker.Device_2_EtherCAT.Term_9_EK1100.Term_35_EL6001.COM_Outputs.Ctrl/Send_continues <-> COM Outputs/Ctrl/Send continues
//     PlcTask Outputs/GVL_iXlinker.Device_2_EtherCAT.Term_9_EK1100.Term_35_EL6001.COM_Outputs.Ctrl/Transmit_request <-> COM Outputs/Ctrl/Transmit request
//     PlcTask Outputs/GVL_iXlinker.Device_2_EtherCAT.Term_9_EK1100.Term_35_EL6001.COM_Outputs.Data_Out[{0..21}] <-> COM Outputs/Data Out {0..21}  (22 links)
//   Plc1/Plc1 Instance <-> Device 2 (EtherCAT)/Term 9 (EK1100)/Term 36 (EL3024)
//     PlcTask Inputs/GVL_iXlinker.Device_2_EtherCAT.Term_9_EK1100.Term_36_EL3024.AI_Standard_Channel_{1..4}.Status/Error <-> AI Standard Channel {1..4}/Status/Error  (4 links)
//     PlcTask Inputs/GVL_iXlinker.Device_2_EtherCAT.Term_9_EK1100.Term_36_EL3024.AI_Standard_Channel_1.Status/Limit_1 <-> AI Standard Channel 1/Status/Limit 1
//     PlcTask Inputs/GVL_iXlinker.Device_2_EtherCAT.Term_9_EK1100.Term_36_EL3024.AI_Standard_Channel_1.Status/Limit_2 <-> AI Standard Channel 1/Status/Limit 2
//     PlcTask Inputs/GVL_iXlinker.Device_2_EtherCAT.Term_9_EK1100.Term_36_EL3024.AI_Standard_Channel_2.Status/Limit_1 <-> AI Standard Channel 2/Status/Limit 1
//     PlcTask Inputs/GVL_iXlinker.Device_2_EtherCAT.Term_9_EK1100.Term_36_EL3024.AI_Standard_Channel_2.Status/Limit_2 <-> AI Standard Channel 2/Status/Limit 2
//     PlcTask Inputs/GVL_iXlinker.Device_2_EtherCAT.Term_9_EK1100.Term_36_EL3024.AI_Standard_Channel_3.Status/Limit_1 <-> AI Standard Channel 3/Status/Limit 1
//     PlcTask Inputs/GVL_iXlinker.Device_2_EtherCAT.Term_9_EK1100.Term_36_EL3024.AI_Standard_Channel_3.Status/Limit_2 <-> AI Standard Channel 3/Status/Limit 2
//     PlcTask Inputs/GVL_iXlinker.Device_2_EtherCAT.Term_9_EK1100.Term_36_EL3024.AI_Standard_Channel_4.Status/Limit_1 <-> AI Standard Channel 4/Status/Limit 1
//     PlcTask Inputs/GVL_iXlinker.Device_2_EtherCAT.Term_9_EK1100.Term_36_EL3024.AI_Standard_Channel_4.Status/Limit_2 <-> AI Standard Channel 4/Status/Limit 2
//     PlcTask Inputs/GVL_iXlinker.Device_2_EtherCAT.Term_9_EK1100.Term_36_EL3024.AI_Standard_Channel_{1..4}.Status/Overrange <-> AI Standard Channel {1..4}/Status/Overrange  (4 links)
//     PlcTask Inputs/GVL_iXlinker.Device_2_EtherCAT.Term_9_EK1100.Term_36_EL3024.AI_Standard_Channel_{1..4}.Status/TxPDO_State <-> AI Standard Channel {1..4}/Status/TxPDO State  (4 links)
//     PlcTask Inputs/GVL_iXlinker.Device_2_EtherCAT.Term_9_EK1100.Term_36_EL3024.AI_Standard_Channel_{1..4}.Status/TxPDO_Toggle <-> AI Standard Channel {1..4}/Status/TxPDO Toggle  (4 links)
//     PlcTask Inputs/GVL_iXlinker.Device_2_EtherCAT.Term_9_EK1100.Term_36_EL3024.AI_Standard_Channel_{1..4}.Status/Underrange <-> AI Standard Channel {1..4}/Status/Underrange  (4 links)
//     PlcTask Inputs/GVL_iXlinker.Device_2_EtherCAT.Term_9_EK1100.Term_36_EL3024.AI_Standard_Channel_{1..4}.Value <-> AI Standard Channel {1..4}/Value  (4 links)
//     PlcTask Inputs/GVL_iXlinker.Device_2_EtherCAT.Term_9_EK1100.Term_36_EL3024.InfoData.AdsAddr <-> InfoData/AdsAddr
//     PlcTask Inputs/GVL_iXlinker.Device_2_EtherCAT.Term_9_EK1100.Term_36_EL3024.InfoData.State <-> InfoData/State
//     PlcTask Inputs/GVL_iXlinker.Device_2_EtherCAT.Term_9_EK1100.Term_36_EL3024.WcState.InputToggle <-> WcState/InputToggle
//     PlcTask Inputs/GVL_iXlinker.Device_2_EtherCAT.Term_9_EK1100.Term_36_EL3024.WcState.WcState <-> WcState/WcState
//   Plc1/Plc1 Instance <-> Device 3 (EtherCAT)
//     PlcTask Inputs/GVL_iXlinker.Device_3_EtherCAT.InfoData.AmsNetId <-> InfoData/AmsNetId
//     PlcTask Inputs/GVL_iXlinker.Device_3_EtherCAT.InfoData.CfgSlaveCount <-> InfoData/CfgSlaveCount
//     PlcTask Inputs/GVL_iXlinker.Device_3_EtherCAT.InfoData.ChangeCount <-> InfoData/ChangeCount
//     PlcTask Inputs/GVL_iXlinker.Device_3_EtherCAT.InfoData.DevId <-> InfoData/DevId
//     PlcTask Inputs/GVL_iXlinker.Device_3_EtherCAT.Inputs.DevState <-> Inputs/DevState
//     PlcTask Inputs/GVL_iXlinker.Device_3_EtherCAT.Inputs.Frm0InputToggle <-> Inputs/Frm0InputToggle
//     PlcTask Inputs/GVL_iXlinker.Device_3_EtherCAT.Inputs.Frm0State <-> Inputs/Frm0State
//     PlcTask Inputs/GVL_iXlinker.Device_3_EtherCAT.Inputs.Frm0WcState <-> Inputs/Frm0WcState
//     PlcTask Inputs/GVL_iXlinker.Device_3_EtherCAT.Inputs.SlaveCount <-> Inputs/SlaveCount
//     PlcTask Inputs/GVL_iXlinker.Device_3_EtherCAT.SyncUnits._default.PlcTask.InfoData.ObjectId <-> SyncUnits/<default>/PlcTask/InfoData/ObjectId
//     PlcTask Inputs/GVL_iXlinker.Device_3_EtherCAT.SyncUnits._default.PlcTask.InfoData.SlaveCount <-> SyncUnits/<default>/PlcTask/InfoData/SlaveCount
//     PlcTask Inputs/GVL_iXlinker.Device_3_EtherCAT.SyncUnits._default.PlcTask.InfoData.State <-> SyncUnits/<default>/PlcTask/InfoData/State
//     PlcTask Inputs/GVL_iXlinker.Device_3_EtherCAT.SyncUnits._default.PlcTask.WcState.WcState <-> SyncUnits/<default>/PlcTask/WcState/WcState
//     PlcTask Outputs/GVL_iXlinker.Device_3_EtherCAT.Outputs.DevCtrl <-> Outputs/DevCtrl
//     PlcTask Outputs/GVL_iXlinker.Device_3_EtherCAT.Outputs.Frm0Ctrl <-> Outputs/Frm0Ctrl
//     PlcTask Outputs/GVL_iXlinker.Device_3_EtherCAT.Outputs.Frm0WcCtrl <-> Outputs/Frm0WcCtrl
//   Plc1/Plc1 Instance <-> Device 3 (EtherCAT)/Term 146 (EK1100)
//     PlcTask Inputs/GVL_iXlinker.Device_3_EtherCAT.Term_146_EK1100.InfoData.State <-> InfoData/State
//   Plc1/Plc1 Instance <-> Device 3 (EtherCAT)/Term 146 (EK1100)/Term 1158 (EL2008)
//     PlcTask Inputs/GVL_iXlinker.Device_3_EtherCAT.Term_146_EK1100.Term_1158_EL2008.InfoData.State <-> InfoData/State
//     PlcTask Inputs/GVL_iXlinker.Device_3_EtherCAT.Term_146_EK1100.Term_1158_EL2008.WcState.WcState <-> WcState/WcState
//     PlcTask Outputs/GVL_iXlinker.Device_3_EtherCAT.Term_146_EK1100.Term_1158_EL2008.Channel_{1..8}.Output <-> Channel {1..8}/Output  (8 links)
//   Plc1/Plc1 Instance <-> Device 3 (EtherCAT)/Term 146 (EK1100)/Term 1159 (EL2008)
//     PlcTask Inputs/GVL_iXlinker.Device_3_EtherCAT.Term_146_EK1100.Term_1159_EL2008.InfoData.State <-> InfoData/State
//     PlcTask Inputs/GVL_iXlinker.Device_3_EtherCAT.Term_146_EK1100.Term_1159_EL2008.WcState.WcState <-> WcState/WcState
//     PlcTask Outputs/GVL_iXlinker.Device_3_EtherCAT.Term_146_EK1100.Term_1159_EL2008.Channel_{1..8}.Output <-> Channel {1..8}/Output  (8 links)
//   Plc1/Plc1 Instance <-> Device 3 (EtherCAT)/Term 146 (EK1100)/Term 1160 (EL2008)
//     PlcTask Inputs/GVL_iXlinker.Device_3_EtherCAT.Term_146_EK1100.Term_1160_EL2008.InfoData.State <-> InfoData/State
//     PlcTask Inputs/GVL_iXlinker.Device_3_EtherCAT.Term_146_EK1100.Term_1160_EL2008.WcState.WcState <-> WcState/WcState
//     PlcTask Outputs/GVL_iXlinker.Device_3_EtherCAT.Term_146_EK1100.Term_1160_EL2008.Channel_{1..8}.Output <-> Channel {1..8}/Output  (8 links)
//   Plc1/Plc1 Instance <-> Device 3 (EtherCAT)/Term 146 (EK1100)/Term 1161 (EL2008)
//     PlcTask Inputs/GVL_iXlinker.Device_3_EtherCAT.Term_146_EK1100.Term_1161_EL2008.InfoData.State <-> InfoData/State
//     PlcTask Inputs/GVL_iXlinker.Device_3_EtherCAT.Term_146_EK1100.Term_1161_EL2008.WcState.WcState <-> WcState/WcState
//     PlcTask Outputs/GVL_iXlinker.Device_3_EtherCAT.Term_146_EK1100.Term_1161_EL2008.Channel_{1..8}.Output <-> Channel {1..8}/Output  (8 links)
//   Plc1/Plc1 Instance <-> Device 3 (EtherCAT)/Term 146 (EK1100)/Term 1162 (EL2008)
//     PlcTask Inputs/GVL_iXlinker.Device_3_EtherCAT.Term_146_EK1100.Term_1162_EL2008.InfoData.State <-> InfoData/State
//     PlcTask Inputs/GVL_iXlinker.Device_3_EtherCAT.Term_146_EK1100.Term_1162_EL2008.WcState.WcState <-> WcState/WcState
//     PlcTask Outputs/GVL_iXlinker.Device_3_EtherCAT.Term_146_EK1100.Term_1162_EL2008.Channel_{1..8}.Output <-> Channel {1..8}/Output  (8 links)
//   Plc1/Plc1 Instance <-> Device 3 (EtherCAT)/Term 146 (EK1100)/Term 1163 (EL2008)
//     PlcTask Inputs/GVL_iXlinker.Device_3_EtherCAT.Term_146_EK1100.Term_1163_EL2008.InfoData.State <-> InfoData/State
//     PlcTask Inputs/GVL_iXlinker.Device_3_EtherCAT.Term_146_EK1100.Term_1163_EL2008.WcState.WcState <-> WcState/WcState
//     PlcTask Outputs/GVL_iXlinker.Device_3_EtherCAT.Term_146_EK1100.Term_1163_EL2008.Channel_{1..8}.Output <-> Channel {1..8}/Output  (8 links)
//   Plc1/Plc1 Instance <-> Device 3 (EtherCAT)/Term 146 (EK1100)/Term 147 (EK1122)
//     PlcTask Inputs/GVL_iXlinker.Device_3_EtherCAT.Term_146_EK1100.Term_147_EK1122.InfoData.State <-> InfoData/State
//   Plc1/Plc1 Instance <-> Device 3 (EtherCAT)/Term 146 (EK1100)/Term 147 (EK1122)/Term 153 (EK1100)
//     PlcTask Inputs/GVL_iXlinker.Device_3_EtherCAT.Term_146_EK1100.Term_147_EK1122.Term_153_EK1100.InfoData.State <-> InfoData/State
//   Plc1/Plc1 Instance <-> Device 3 (EtherCAT)/Term 146 (EK1100)/Term 147 (EK1122)/Term 153 (EK1100)/Term 154 (EK1122)
//     PlcTask Inputs/GVL_iXlinker.Device_3_EtherCAT.Term_146_EK1100.Term_147_EK1122.Term_153_EK1100.Term_154_EK1122.InfoData.State <-> InfoData/State
//   Plc1/Plc1 Instance <-> Device 3 (EtherCAT)/Term 146 (EK1100)/Term 147 (EK1122)/Term 153 (EK1100)/Term 154 (EK1122)/Term 157 (EK1100)
//     PlcTask Inputs/GVL_iXlinker.Device_3_EtherCAT.Term_146_EK1100.Term_147_EK1122.Term_153_EK1100.Term_154_EK1122.Term_157_EK1100.InfoData.State <-> InfoData/State
//   Plc1/Plc1 Instance <-> Device 3 (EtherCAT)/Term 146 (EK1100)/Term 147 (EK1122)/Term 153 (EK1100)/Term 154 (EK1122)/Term 157 (EK1100)/Term 159 (EL1809)
//     PlcTask Inputs/GVL_iXlinker.Device_3_EtherCAT.Term_146_EK1100.Term_147_EK1122.Term_153_EK1100.Term_154_EK1122.Term_157_EK1100.Term_159_EL1809.Channel_{1..16}.Input <-> Channel {1..16}/Input  (16 links)
//     PlcTask Inputs/GVL_iXlinker.Device_3_EtherCAT.Term_146_EK1100.Term_147_EK1122.Term_153_EK1100.Term_154_EK1122.Term_157_EK1100.Term_159_EL1809.InfoData.State <-> InfoData/State
//     PlcTask Inputs/GVL_iXlinker.Device_3_EtherCAT.Term_146_EK1100.Term_147_EK1122.Term_153_EK1100.Term_154_EK1122.Term_157_EK1100.Term_159_EL1809.WcState.InputToggle <-> WcState/InputToggle
//     PlcTask Inputs/GVL_iXlinker.Device_3_EtherCAT.Term_146_EK1100.Term_147_EK1122.Term_153_EK1100.Term_154_EK1122.Term_157_EK1100.Term_159_EL1809.WcState.WcState <-> WcState/WcState
//   Plc1/Plc1 Instance <-> Device 3 (EtherCAT)/Term 146 (EK1100)/Term 147 (EK1122)/Term 153 (EK1100)/Term 154 (EK1122)/Term 158 (EK1100)
//     PlcTask Inputs/GVL_iXlinker.Device_3_EtherCAT.Term_146_EK1100.Term_147_EK1122.Term_153_EK1100.Term_154_EK1122.Term_158_EK1100.InfoData.State <-> InfoData/State
//   Plc1/Plc1 Instance <-> Device 3 (EtherCAT)/Term 146 (EK1100)/Term 147 (EK1122)/Term 153 (EK1100)/Term 154 (EK1122)/Term 158 (EK1100)/Term 160 (EL1809)
//     PlcTask Inputs/GVL_iXlinker.Device_3_EtherCAT.Term_146_EK1100.Term_147_EK1122.Term_153_EK1100.Term_154_EK1122.Term_158_EK1100.Term_160_EL1809.Channel_{1..16}.Input <-> Channel {1..16}/Input  (16 links)
//     PlcTask Inputs/GVL_iXlinker.Device_3_EtherCAT.Term_146_EK1100.Term_147_EK1122.Term_153_EK1100.Term_154_EK1122.Term_158_EK1100.Term_160_EL1809.InfoData.State <-> InfoData/State
//     PlcTask Inputs/GVL_iXlinker.Device_3_EtherCAT.Term_146_EK1100.Term_147_EK1122.Term_153_EK1100.Term_154_EK1122.Term_158_EK1100.Term_160_EL1809.WcState.InputToggle <-> WcState/InputToggle
//     PlcTask Inputs/GVL_iXlinker.Device_3_EtherCAT.Term_146_EK1100.Term_147_EK1122.Term_153_EK1100.Term_154_EK1122.Term_158_EK1100.Term_160_EL1809.WcState.WcState <-> WcState/WcState
//   Plc1/Plc1 Instance <-> Device 3 (EtherCAT)/Term 146 (EK1100)/Term 147 (EK1122)/Term 153 (EK1100)/Term 155 (EL2008)
//     PlcTask Inputs/GVL_iXlinker.Device_3_EtherCAT.Term_146_EK1100.Term_147_EK1122.Term_153_EK1100.Term_155_EL2008.InfoData.State <-> InfoData/State
//     PlcTask Inputs/GVL_iXlinker.Device_3_EtherCAT.Term_146_EK1100.Term_147_EK1122.Term_153_EK1100.Term_155_EL2008.WcState.WcState <-> WcState/WcState
//     PlcTask Outputs/GVL_iXlinker.Device_3_EtherCAT.Term_146_EK1100.Term_147_EK1122.Term_153_EK1100.Term_155_EL2008.Channel_{1..8}.Output <-> Channel {1..8}/Output  (8 links)
//   Plc1/Plc1 Instance <-> Device 3 (EtherCAT)/Term 146 (EK1100)/Term 147 (EK1122)/Term 153 (EK1100)/Term 156 (EL2008)
//     PlcTask Inputs/GVL_iXlinker.Device_3_EtherCAT.Term_146_EK1100.Term_147_EK1122.Term_153_EK1100.Term_156_EL2008.InfoData.State <-> InfoData/State
//     PlcTask Inputs/GVL_iXlinker.Device_3_EtherCAT.Term_146_EK1100.Term_147_EK1122.Term_153_EK1100.Term_156_EL2008.WcState.WcState <-> WcState/WcState
//     PlcTask Outputs/GVL_iXlinker.Device_3_EtherCAT.Term_146_EK1100.Term_147_EK1122.Term_153_EK1100.Term_156_EL2008.Channel_{1..8}.Output <-> Channel {1..8}/Output  (8 links)
//   Plc1/Plc1 Instance <-> Device 3 (EtherCAT)/Term 146 (EK1100)/Term 147 (EK1122)/Term 178 (EK1100)
//     PlcTask Inputs/GVL_iXlinker.Device_3_EtherCAT.Term_146_EK1100.Term_147_EK1122.Term_178_EK1100.InfoData.State <-> InfoData/State
//   Plc1/Plc1 Instance <-> Device 3 (EtherCAT)/Term 146 (EK1100)/Term 147 (EK1122)/Term 178 (EK1100)/Term 179 (EK1122)
//     PlcTask Inputs/GVL_iXlinker.Device_3_EtherCAT.Term_146_EK1100.Term_147_EK1122.Term_178_EK1100.Term_179_EK1122.InfoData.State <-> InfoData/State
//   Plc1/Plc1 Instance <-> Device 3 (EtherCAT)/Term 146 (EK1100)/Term 147 (EK1122)/Term 178 (EK1100)/Term 179 (EK1122)/Term 180 (EK1100)
//     PlcTask Inputs/GVL_iXlinker.Device_3_EtherCAT.Term_146_EK1100.Term_147_EK1122.Term_178_EK1100.Term_179_EK1122.Term_180_EK1100.InfoData.State <-> InfoData/State
//   Plc1/Plc1 Instance <-> Device 3 (EtherCAT)/Term 146 (EK1100)/Term 147 (EK1122)/Term 178 (EK1100)/Term 179 (EK1122)/Term 180 (EK1100)/Term 181 (EL1809)
//     PlcTask Inputs/GVL_iXlinker.Device_3_EtherCAT.Term_146_EK1100.Term_147_EK1122.Term_178_EK1100.Term_179_EK1122.Term_180_EK1100.Term_181_EL1809.Channel_{1..16}.Input <-> Channel {1..16}/Input  (16 links)
//     PlcTask Inputs/GVL_iXlinker.Device_3_EtherCAT.Term_146_EK1100.Term_147_EK1122.Term_178_EK1100.Term_179_EK1122.Term_180_EK1100.Term_181_EL1809.InfoData.State <-> InfoData/State
//     PlcTask Inputs/GVL_iXlinker.Device_3_EtherCAT.Term_146_EK1100.Term_147_EK1122.Term_178_EK1100.Term_179_EK1122.Term_180_EK1100.Term_181_EL1809.WcState.InputToggle <-> WcState/InputToggle
//     PlcTask Inputs/GVL_iXlinker.Device_3_EtherCAT.Term_146_EK1100.Term_147_EK1122.Term_178_EK1100.Term_179_EK1122.Term_180_EK1100.Term_181_EL1809.WcState.WcState <-> WcState/WcState
//   Plc1/Plc1 Instance <-> Device 3 (EtherCAT)/Term 146 (EK1100)/Term 147 (EK1122)/Term 178 (EK1100)/Term 179 (EK1122)/Term 182 (EK1100)
//     PlcTask Inputs/GVL_iXlinker.Device_3_EtherCAT.Term_146_EK1100.Term_147_EK1122.Term_178_EK1100.Term_179_EK1122.Term_182_EK1100.InfoData.State <-> InfoData/State
//   Plc1/Plc1 Instance <-> Device 3 (EtherCAT)/Term 146 (EK1100)/Term 147 (EK1122)/Term 178 (EK1100)/Term 179 (EK1122)/Term 182 (EK1100)/Term 183 (EL1809)
//     PlcTask Inputs/GVL_iXlinker.Device_3_EtherCAT.Term_146_EK1100.Term_147_EK1122.Term_178_EK1100.Term_179_EK1122.Term_182_EK1100.Term_183_EL1809.Channel_{1..16}.Input <-> Channel {1..16}/Input  (16 links)
//     PlcTask Inputs/GVL_iXlinker.Device_3_EtherCAT.Term_146_EK1100.Term_147_EK1122.Term_178_EK1100.Term_179_EK1122.Term_182_EK1100.Term_183_EL1809.InfoData.State <-> InfoData/State
//     PlcTask Inputs/GVL_iXlinker.Device_3_EtherCAT.Term_146_EK1100.Term_147_EK1122.Term_178_EK1100.Term_179_EK1122.Term_182_EK1100.Term_183_EL1809.WcState.InputToggle <-> WcState/InputToggle
//     PlcTask Inputs/GVL_iXlinker.Device_3_EtherCAT.Term_146_EK1100.Term_147_EK1122.Term_178_EK1100.Term_179_EK1122.Term_182_EK1100.Term_183_EL1809.WcState.WcState <-> WcState/WcState
//   Plc1/Plc1 Instance <-> Device 3 (EtherCAT)/Term 146 (EK1100)/Term 147 (EK1122)/Term 178 (EK1100)/Term 184 (EL2008)
//     PlcTask Inputs/GVL_iXlinker.Device_3_EtherCAT.Term_146_EK1100.Term_147_EK1122.Term_178_EK1100.Term_184_EL2008.InfoData.State <-> InfoData/State
//     PlcTask Inputs/GVL_iXlinker.Device_3_EtherCAT.Term_146_EK1100.Term_147_EK1122.Term_178_EK1100.Term_184_EL2008.WcState.WcState <-> WcState/WcState
//     PlcTask Outputs/GVL_iXlinker.Device_3_EtherCAT.Term_146_EK1100.Term_147_EK1122.Term_178_EK1100.Term_184_EL2008.Channel_{1..8}.Output <-> Channel {1..8}/Output  (8 links)
//   Plc1/Plc1 Instance <-> Device 3 (EtherCAT)/Term 146 (EK1100)/Term 147 (EK1122)/Term 178 (EK1100)/Term 185 (EL2008)
//     PlcTask Inputs/GVL_iXlinker.Device_3_EtherCAT.Term_146_EK1100.Term_147_EK1122.Term_178_EK1100.Term_185_EL2008.InfoData.State <-> InfoData/State
//     PlcTask Inputs/GVL_iXlinker.Device_3_EtherCAT.Term_146_EK1100.Term_147_EK1122.Term_178_EK1100.Term_185_EL2008.WcState.WcState <-> WcState/WcState
//     PlcTask Outputs/GVL_iXlinker.Device_3_EtherCAT.Term_146_EK1100.Term_147_EK1122.Term_178_EK1100.Term_185_EL2008.Channel_{1..8}.Output <-> Channel {1..8}/Output  (8 links)
//   Plc1/Plc1 Instance <-> Device 3 (EtherCAT)/Term 146 (EK1100)/Term 148 (EL1809)
//     PlcTask Inputs/GVL_iXlinker.Device_3_EtherCAT.Term_146_EK1100.Term_148_EL1809.Channel_{1..16}.Input <-> Channel {1..16}/Input  (16 links)
//     PlcTask Inputs/GVL_iXlinker.Device_3_EtherCAT.Term_146_EK1100.Term_148_EL1809.InfoData.State <-> InfoData/State
//     PlcTask Inputs/GVL_iXlinker.Device_3_EtherCAT.Term_146_EK1100.Term_148_EL1809.WcState.InputToggle <-> WcState/InputToggle
//     PlcTask Inputs/GVL_iXlinker.Device_3_EtherCAT.Term_146_EK1100.Term_148_EL1809.WcState.WcState <-> WcState/WcState
//   Plc1/Plc1 Instance <-> Device 3 (EtherCAT)/Term 146 (EK1100)/Term 149 (EL1809)
//     PlcTask Inputs/GVL_iXlinker.Device_3_EtherCAT.Term_146_EK1100.Term_149_EL1809.Channel_{1..16}.Input <-> Channel {1..16}/Input  (16 links)
//     PlcTask Inputs/GVL_iXlinker.Device_3_EtherCAT.Term_146_EK1100.Term_149_EL1809.InfoData.State <-> InfoData/State
//     PlcTask Inputs/GVL_iXlinker.Device_3_EtherCAT.Term_146_EK1100.Term_149_EL1809.WcState.InputToggle <-> WcState/InputToggle
//     PlcTask Inputs/GVL_iXlinker.Device_3_EtherCAT.Term_146_EK1100.Term_149_EL1809.WcState.WcState <-> WcState/WcState
//   Plc1/Plc1 Instance <-> Device 3 (EtherCAT)/Term 146 (EK1100)/Term 150 (EL1809)
//     PlcTask Inputs/GVL_iXlinker.Device_3_EtherCAT.Term_146_EK1100.Term_150_EL1809.Channel_{1..16}.Input <-> Channel {1..16}/Input  (16 links)
//     PlcTask Inputs/GVL_iXlinker.Device_3_EtherCAT.Term_146_EK1100.Term_150_EL1809.InfoData.State <-> InfoData/State
//     PlcTask Inputs/GVL_iXlinker.Device_3_EtherCAT.Term_146_EK1100.Term_150_EL1809.WcState.InputToggle <-> WcState/InputToggle
//     PlcTask Inputs/GVL_iXlinker.Device_3_EtherCAT.Term_146_EK1100.Term_150_EL1809.WcState.WcState <-> WcState/WcState
//   Plc1/Plc1 Instance <-> Device 3 (EtherCAT)/Term 146 (EK1100)/Term 151 (EL1809)
//     PlcTask Inputs/GVL_iXlinker.Device_3_EtherCAT.Term_146_EK1100.Term_151_EL1809.Channel_{1..16}.Input <-> Channel {1..16}/Input  (16 links)
//     PlcTask Inputs/GVL_iXlinker.Device_3_EtherCAT.Term_146_EK1100.Term_151_EL1809.InfoData.State <-> InfoData/State
//     PlcTask Inputs/GVL_iXlinker.Device_3_EtherCAT.Term_146_EK1100.Term_151_EL1809.WcState.InputToggle <-> WcState/InputToggle
//     PlcTask Inputs/GVL_iXlinker.Device_3_EtherCAT.Term_146_EK1100.Term_151_EL1809.WcState.WcState <-> WcState/WcState
//   Plc1/Plc1 Instance <-> Device 3 (EtherCAT)/Term 146 (EK1100)/Term 152 (EL1809)
//     PlcTask Inputs/GVL_iXlinker.Device_3_EtherCAT.Term_146_EK1100.Term_152_EL1809.Channel_{1..16}.Input <-> Channel {1..16}/Input  (16 links)
//     PlcTask Inputs/GVL_iXlinker.Device_3_EtherCAT.Term_146_EK1100.Term_152_EL1809.InfoData.State <-> InfoData/State
//     PlcTask Inputs/GVL_iXlinker.Device_3_EtherCAT.Term_146_EK1100.Term_152_EL1809.WcState.InputToggle <-> WcState/InputToggle
//     PlcTask Inputs/GVL_iXlinker.Device_3_EtherCAT.Term_146_EK1100.Term_152_EL1809.WcState.WcState <-> WcState/WcState
//   Plc1/Plc1 Instance <-> Device 3 (EtherCAT)/Term 146 (EK1100)/Term 186 (EK1122)
//     PlcTask Inputs/GVL_iXlinker.Device_3_EtherCAT.Term_146_EK1100.Term_186_EK1122.InfoData.State <-> InfoData/State
//   Plc1/Plc1 Instance <-> Device 3 (EtherCAT)/Term 146 (EK1100)/Term 186 (EK1122)/Term 187 (EK1100)
//     PlcTask Inputs/GVL_iXlinker.Device_3_EtherCAT.Term_146_EK1100.Term_186_EK1122.Term_187_EK1100.InfoData.State <-> InfoData/State
//   Plc1/Plc1 Instance <-> Device 3 (EtherCAT)/Term 146 (EK1100)/Term 186 (EK1122)/Term 187 (EK1100)/Term 188 (EK1122)
//     PlcTask Inputs/GVL_iXlinker.Device_3_EtherCAT.Term_146_EK1100.Term_186_EK1122.Term_187_EK1100.Term_188_EK1122.InfoData.State <-> InfoData/State
//   Plc1/Plc1 Instance <-> Device 3 (EtherCAT)/Term 146 (EK1100)/Term 186 (EK1122)/Term 187 (EK1100)/Term 188 (EK1122)/Term 189 (EK1100)
//     PlcTask Inputs/GVL_iXlinker.Device_3_EtherCAT.Term_146_EK1100.Term_186_EK1122.Term_187_EK1100.Term_188_EK1122.Term_189_EK1100.InfoData.State <-> InfoData/State
//   Plc1/Plc1 Instance <-> Device 3 (EtherCAT)/Term 146 (EK1100)/Term 186 (EK1122)/Term 187 (EK1100)/Term 188 (EK1122)/Term 189 (EK1100)/Term 193 (EL1809)
//     PlcTask Inputs/GVL_iXlinker.Device_3_EtherCAT.Term_146_EK1100.Term_186_EK1122.Term_187_EK1100.Term_188_EK1122.Term_189_EK1100.Term_193_EL1809.Channel_{1..16}.Input <-> Channel {1..16}/Input  (16 links)
//     PlcTask Inputs/GVL_iXlinker.Device_3_EtherCAT.Term_146_EK1100.Term_186_EK1122.Term_187_EK1100.Term_188_EK1122.Term_189_EK1100.Term_193_EL1809.InfoData.State <-> InfoData/State
//     PlcTask Inputs/GVL_iXlinker.Device_3_EtherCAT.Term_146_EK1100.Term_186_EK1122.Term_187_EK1100.Term_188_EK1122.Term_189_EK1100.Term_193_EL1809.WcState.InputToggle <-> WcState/InputToggle
//     PlcTask Inputs/GVL_iXlinker.Device_3_EtherCAT.Term_146_EK1100.Term_186_EK1122.Term_187_EK1100.Term_188_EK1122.Term_189_EK1100.Term_193_EL1809.WcState.WcState <-> WcState/WcState
//   Plc1/Plc1 Instance <-> Device 3 (EtherCAT)/Term 146 (EK1100)/Term 186 (EK1122)/Term 187 (EK1100)/Term 188 (EK1122)/Term 194 (EK1100)
//     PlcTask Inputs/GVL_iXlinker.Device_3_EtherCAT.Term_146_EK1100.Term_186_EK1122.Term_187_EK1100.Term_188_EK1122.Term_194_EK1100.InfoData.State <-> InfoData/State
//   Plc1/Plc1 Instance <-> Device 3 (EtherCAT)/Term 146 (EK1100)/Term 186 (EK1122)/Term 187 (EK1100)/Term 188 (EK1122)/Term 194 (EK1100)/Term 200 (EL1809)
//     PlcTask Inputs/GVL_iXlinker.Device_3_EtherCAT.Term_146_EK1100.Term_186_EK1122.Term_187_EK1100.Term_188_EK1122.Term_194_EK1100.Term_200_EL1809.Channel_{1..16}.Input <-> Channel {1..16}/Input  (16 links)
//     PlcTask Inputs/GVL_iXlinker.Device_3_EtherCAT.Term_146_EK1100.Term_186_EK1122.Term_187_EK1100.Term_188_EK1122.Term_194_EK1100.Term_200_EL1809.InfoData.State <-> InfoData/State
//     PlcTask Inputs/GVL_iXlinker.Device_3_EtherCAT.Term_146_EK1100.Term_186_EK1122.Term_187_EK1100.Term_188_EK1122.Term_194_EK1100.Term_200_EL1809.WcState.InputToggle <-> WcState/InputToggle
//     PlcTask Inputs/GVL_iXlinker.Device_3_EtherCAT.Term_146_EK1100.Term_186_EK1122.Term_187_EK1100.Term_188_EK1122.Term_194_EK1100.Term_200_EL1809.WcState.WcState <-> WcState/WcState
//   Plc1/Plc1 Instance <-> Device 3 (EtherCAT)/Term 146 (EK1100)/Term 186 (EK1122)/Term 187 (EK1100)/Term 204 (EL2008)
//     PlcTask Inputs/GVL_iXlinker.Device_3_EtherCAT.Term_146_EK1100.Term_186_EK1122.Term_187_EK1100.Term_204_EL2008.InfoData.State <-> InfoData/State
//     PlcTask Inputs/GVL_iXlinker.Device_3_EtherCAT.Term_146_EK1100.Term_186_EK1122.Term_187_EK1100.Term_204_EL2008.WcState.WcState <-> WcState/WcState
//     PlcTask Outputs/GVL_iXlinker.Device_3_EtherCAT.Term_146_EK1100.Term_186_EK1122.Term_187_EK1100.Term_204_EL2008.Channel_{1..8}.Output <-> Channel {1..8}/Output  (8 links)
//   Plc1/Plc1 Instance <-> Device 3 (EtherCAT)/Term 146 (EK1100)/Term 186 (EK1122)/Term 187 (EK1100)/Term 205 (EL2008)
//     PlcTask Inputs/GVL_iXlinker.Device_3_EtherCAT.Term_146_EK1100.Term_186_EK1122.Term_187_EK1100.Term_205_EL2008.InfoData.State <-> InfoData/State
//     PlcTask Inputs/GVL_iXlinker.Device_3_EtherCAT.Term_146_EK1100.Term_186_EK1122.Term_187_EK1100.Term_205_EL2008.WcState.WcState <-> WcState/WcState
//     PlcTask Outputs/GVL_iXlinker.Device_3_EtherCAT.Term_146_EK1100.Term_186_EK1122.Term_187_EK1100.Term_205_EL2008.Channel_{1..8}.Output <-> Channel {1..8}/Output  (8 links)
//   Plc1/Plc1 Instance <-> Device 3 (EtherCAT)/Term 146 (EK1100)/Term 186 (EK1122)/Term 207 (EK1100)
//     PlcTask Inputs/GVL_iXlinker.Device_3_EtherCAT.Term_146_EK1100.Term_186_EK1122.Term_207_EK1100.InfoData.State <-> InfoData/State
//   Plc1/Plc1 Instance <-> Device 3 (EtherCAT)/Term 146 (EK1100)/Term 186 (EK1122)/Term 207 (EK1100)/Term 230 (EK1122)
//     PlcTask Inputs/GVL_iXlinker.Device_3_EtherCAT.Term_146_EK1100.Term_186_EK1122.Term_207_EK1100.Term_230_EK1122.InfoData.State <-> InfoData/State
//   Plc1/Plc1 Instance <-> Device 3 (EtherCAT)/Term 146 (EK1100)/Term 186 (EK1122)/Term 207 (EK1100)/Term 230 (EK1122)/Term 231 (EK1100)
//     PlcTask Inputs/GVL_iXlinker.Device_3_EtherCAT.Term_146_EK1100.Term_186_EK1122.Term_207_EK1100.Term_230_EK1122.Term_231_EK1100.InfoData.State <-> InfoData/State
//   Plc1/Plc1 Instance <-> Device 3 (EtherCAT)/Term 146 (EK1100)/Term 186 (EK1122)/Term 207 (EK1100)/Term 230 (EK1122)/Term 231 (EK1100)/Term 232 (EL1809)
//     PlcTask Inputs/GVL_iXlinker.Device_3_EtherCAT.Term_146_EK1100.Term_186_EK1122.Term_207_EK1100.Term_230_EK1122.Term_231_EK1100.Term_232_EL1809.Channel_{1..16}.Input <-> Channel {1..16}/Input  (16 links)
//     PlcTask Inputs/GVL_iXlinker.Device_3_EtherCAT.Term_146_EK1100.Term_186_EK1122.Term_207_EK1100.Term_230_EK1122.Term_231_EK1100.Term_232_EL1809.InfoData.State <-> InfoData/State
//     PlcTask Inputs/GVL_iXlinker.Device_3_EtherCAT.Term_146_EK1100.Term_186_EK1122.Term_207_EK1100.Term_230_EK1122.Term_231_EK1100.Term_232_EL1809.WcState.InputToggle <-> WcState/InputToggle
//     PlcTask Inputs/GVL_iXlinker.Device_3_EtherCAT.Term_146_EK1100.Term_186_EK1122.Term_207_EK1100.Term_230_EK1122.Term_231_EK1100.Term_232_EL1809.WcState.WcState <-> WcState/WcState
//   Plc1/Plc1 Instance <-> Device 3 (EtherCAT)/Term 146 (EK1100)/Term 186 (EK1122)/Term 207 (EK1100)/Term 230 (EK1122)/Term 233 (EK1100)
//     PlcTask Inputs/GVL_iXlinker.Device_3_EtherCAT.Term_146_EK1100.Term_186_EK1122.Term_207_EK1100.Term_230_EK1122.Term_233_EK1100.InfoData.State <-> InfoData/State
//   Plc1/Plc1 Instance <-> Device 3 (EtherCAT)/Term 146 (EK1100)/Term 186 (EK1122)/Term 207 (EK1100)/Term 230 (EK1122)/Term 233 (EK1100)/Term 234 (EL1809)
//     PlcTask Inputs/GVL_iXlinker.Device_3_EtherCAT.Term_146_EK1100.Term_186_EK1122.Term_207_EK1100.Term_230_EK1122.Term_233_EK1100.Term_234_EL1809.Channel_{1..16}.Input <-> Channel {1..16}/Input  (16 links)
//     PlcTask Inputs/GVL_iXlinker.Device_3_EtherCAT.Term_146_EK1100.Term_186_EK1122.Term_207_EK1100.Term_230_EK1122.Term_233_EK1100.Term_234_EL1809.InfoData.State <-> InfoData/State
//     PlcTask Inputs/GVL_iXlinker.Device_3_EtherCAT.Term_146_EK1100.Term_186_EK1122.Term_207_EK1100.Term_230_EK1122.Term_233_EK1100.Term_234_EL1809.WcState.InputToggle <-> WcState/InputToggle
//     PlcTask Inputs/GVL_iXlinker.Device_3_EtherCAT.Term_146_EK1100.Term_186_EK1122.Term_207_EK1100.Term_230_EK1122.Term_233_EK1100.Term_234_EL1809.WcState.WcState <-> WcState/WcState
//   Plc1/Plc1 Instance <-> Device 3 (EtherCAT)/Term 146 (EK1100)/Term 186 (EK1122)/Term 207 (EK1100)/Term 235 (EL2008)
//     PlcTask Inputs/GVL_iXlinker.Device_3_EtherCAT.Term_146_EK1100.Term_186_EK1122.Term_207_EK1100.Term_235_EL2008.InfoData.State <-> InfoData/State
//     PlcTask Inputs/GVL_iXlinker.Device_3_EtherCAT.Term_146_EK1100.Term_186_EK1122.Term_207_EK1100.Term_235_EL2008.WcState.WcState <-> WcState/WcState
//     PlcTask Outputs/GVL_iXlinker.Device_3_EtherCAT.Term_146_EK1100.Term_186_EK1122.Term_207_EK1100.Term_235_EL2008.Channel_{1..8}.Output <-> Channel {1..8}/Output  (8 links)
//   Plc1/Plc1 Instance <-> Device 3 (EtherCAT)/Term 146 (EK1100)/Term 186 (EK1122)/Term 207 (EK1100)/Term 236 (EL2008)
//     PlcTask Inputs/GVL_iXlinker.Device_3_EtherCAT.Term_146_EK1100.Term_186_EK1122.Term_207_EK1100.Term_236_EL2008.InfoData.State <-> InfoData/State
//     PlcTask Inputs/GVL_iXlinker.Device_3_EtherCAT.Term_146_EK1100.Term_186_EK1122.Term_207_EK1100.Term_236_EL2008.WcState.WcState <-> WcState/WcState
//     PlcTask Outputs/GVL_iXlinker.Device_3_EtherCAT.Term_146_EK1100.Term_186_EK1122.Term_207_EK1100.Term_236_EL2008.Channel_{1..8}.Output <-> Channel {1..8}/Output  (8 links)
//   Plc1/Plc1 Instance <-> Device 3 (EtherCAT)/Term 146 (EK1100)/Term 288 (EK1122)
//     PlcTask Inputs/GVL_iXlinker.Device_3_EtherCAT.Term_146_EK1100.Term_288_EK1122.InfoData.State <-> InfoData/State
//   Plc1/Plc1 Instance <-> Device 3 (EtherCAT)/Term 146 (EK1100)/Term 288 (EK1122)/Term 289 (EK1100)
//     PlcTask Inputs/GVL_iXlinker.Device_3_EtherCAT.Term_146_EK1100.Term_288_EK1122.Term_289_EK1100.InfoData.State <-> InfoData/State
//   Plc1/Plc1 Instance <-> Device 3 (EtherCAT)/Term 146 (EK1100)/Term 288 (EK1122)/Term 289 (EK1100)/Term 237 (EK1122)
//     PlcTask Inputs/GVL_iXlinker.Device_3_EtherCAT.Term_146_EK1100.Term_288_EK1122.Term_289_EK1100.Term_237_EK1122.InfoData.State <-> InfoData/State
//   Plc1/Plc1 Instance <-> Device 3 (EtherCAT)/Term 146 (EK1100)/Term 288 (EK1122)/Term 289 (EK1100)/Term 237 (EK1122)/Drive 238 (AX5101-0000-0214)
//     PlcTask Inputs/GVL_iXlinker.Device_3_EtherCAT.Term_146_EK1100.Term_288_EK1122.Term_289_EK1100.Term_237_EK1122.Drive_238_AX5101_0000_0214.AT_x.Drive_status_word <-> AT/Drive status word
//     PlcTask Inputs/GVL_iXlinker.Device_3_EtherCAT.Term_146_EK1100.Term_288_EK1122.Term_289_EK1100.Term_237_EK1122.Drive_238_AX5101_0000_0214.AT_x.Following_distance <-> AT/Following distance
//     PlcTask Inputs/GVL_iXlinker.Device_3_EtherCAT.Term_146_EK1100.Term_288_EK1122.Term_289_EK1100.Term_237_EK1122.Drive_238_AX5101_0000_0214.AT_x.Position_feedback_1_value <-> AT/Position feedback 1 value
//     PlcTask Inputs/GVL_iXlinker.Device_3_EtherCAT.Term_146_EK1100.Term_288_EK1122.Term_289_EK1100.Term_237_EK1122.Drive_238_AX5101_0000_0214.InfoData.AdsAddr <-> InfoData/AdsAddr
//     PlcTask Inputs/GVL_iXlinker.Device_3_EtherCAT.Term_146_EK1100.Term_288_EK1122.Term_289_EK1100.Term_237_EK1122.Drive_238_AX5101_0000_0214.InfoData.Chn0 <-> InfoData/Chn0
//     PlcTask Inputs/GVL_iXlinker.Device_3_EtherCAT.Term_146_EK1100.Term_288_EK1122.Term_289_EK1100.Term_237_EK1122.Drive_238_AX5101_0000_0214.InfoData.DcInputShift <-> InfoData/DcInputShift
//     PlcTask Inputs/GVL_iXlinker.Device_3_EtherCAT.Term_146_EK1100.Term_288_EK1122.Term_289_EK1100.Term_237_EK1122.Drive_238_AX5101_0000_0214.InfoData.DcOutputShift <-> InfoData/DcOutputShift
//     PlcTask Inputs/GVL_iXlinker.Device_3_EtherCAT.Term_146_EK1100.Term_288_EK1122.Term_289_EK1100.Term_237_EK1122.Drive_238_AX5101_0000_0214.InfoData.State <-> InfoData/State
//     PlcTask Inputs/GVL_iXlinker.Device_3_EtherCAT.Term_146_EK1100.Term_288_EK1122.Term_289_EK1100.Term_237_EK1122.Drive_238_AX5101_0000_0214.WcState.InputToggle <-> WcState/InputToggle
//     PlcTask Inputs/GVL_iXlinker.Device_3_EtherCAT.Term_146_EK1100.Term_288_EK1122.Term_289_EK1100.Term_237_EK1122.Drive_238_AX5101_0000_0214.WcState.WcState <-> WcState/WcState
//     PlcTask Outputs/GVL_iXlinker.Device_3_EtherCAT.Term_146_EK1100.Term_288_EK1122.Term_289_EK1100.Term_237_EK1122.Drive_238_AX5101_0000_0214.MDT.Master_control_word <-> MDT/Master control word
//     PlcTask Outputs/GVL_iXlinker.Device_3_EtherCAT.Term_146_EK1100.Term_288_EK1122.Term_289_EK1100.Term_237_EK1122.Drive_238_AX5101_0000_0214.MDT.Position_command_value <-> MDT/Position command value
//   Plc1/Plc1 Instance <-> Device 3 (EtherCAT)/Term 146 (EK1100)/Term 288 (EK1122)/Term 289 (EK1100)/Term 293 (EL1809)
//     PlcTask Inputs/GVL_iXlinker.Device_3_EtherCAT.Term_146_EK1100.Term_288_EK1122.Term_289_EK1100.Term_293_EL1809.Channel_{1..16}.Input <-> Channel {1..16}/Input  (16 links)
//     PlcTask Inputs/GVL_iXlinker.Device_3_EtherCAT.Term_146_EK1100.Term_288_EK1122.Term_289_EK1100.Term_293_EL1809.InfoData.State <-> InfoData/State
//     PlcTask Inputs/GVL_iXlinker.Device_3_EtherCAT.Term_146_EK1100.Term_288_EK1122.Term_289_EK1100.Term_293_EL1809.WcState.InputToggle <-> WcState/InputToggle
//     PlcTask Inputs/GVL_iXlinker.Device_3_EtherCAT.Term_146_EK1100.Term_288_EK1122.Term_289_EK1100.Term_293_EL1809.WcState.WcState <-> WcState/WcState
//   Plc1/Plc1 Instance <-> Device 3 (EtherCAT)/Term 146 (EK1100)/Term 288 (EK1122)/Term 294 (EK1100)
//     PlcTask Inputs/GVL_iXlinker.Device_3_EtherCAT.Term_146_EK1100.Term_288_EK1122.Term_294_EK1100.InfoData.State <-> InfoData/State
//   Plc1/Plc1 Instance <-> Device 3 (EtherCAT)/Term 146 (EK1100)/Term 288 (EK1122)/Term 294 (EK1100)/Term 300 (EL1809)
//     PlcTask Inputs/GVL_iXlinker.Device_3_EtherCAT.Term_146_EK1100.Term_288_EK1122.Term_294_EK1100.Term_300_EL1809.Channel_{1..16}.Input <-> Channel {1..16}/Input  (16 links)
//     PlcTask Inputs/GVL_iXlinker.Device_3_EtherCAT.Term_146_EK1100.Term_288_EK1122.Term_294_EK1100.Term_300_EL1809.InfoData.State <-> InfoData/State
//     PlcTask Inputs/GVL_iXlinker.Device_3_EtherCAT.Term_146_EK1100.Term_288_EK1122.Term_294_EK1100.Term_300_EL1809.WcState.InputToggle <-> WcState/InputToggle
//     PlcTask Inputs/GVL_iXlinker.Device_3_EtherCAT.Term_146_EK1100.Term_288_EK1122.Term_294_EK1100.Term_300_EL1809.WcState.WcState <-> WcState/WcState
//   Plc1/Plc1 Instance <-> Device 3 (EtherCAT)/Term 146 (EK1100)/Term 288 (EK1122)/Term 294 (EK1100)/Term 304 (EL2008)
//     PlcTask Inputs/GVL_iXlinker.Device_3_EtherCAT.Term_146_EK1100.Term_288_EK1122.Term_294_EK1100.Term_304_EL2008.InfoData.State <-> InfoData/State
//     PlcTask Inputs/GVL_iXlinker.Device_3_EtherCAT.Term_146_EK1100.Term_288_EK1122.Term_294_EK1100.Term_304_EL2008.WcState.WcState <-> WcState/WcState
//     PlcTask Outputs/GVL_iXlinker.Device_3_EtherCAT.Term_146_EK1100.Term_288_EK1122.Term_294_EK1100.Term_304_EL2008.Channel_{1..8}.Output <-> Channel {1..8}/Output  (8 links)
//   Plc1/Plc1 Instance <-> Device 3 (EtherCAT)/Term 146 (EK1100)/Term 288 (EK1122)/Term 294 (EK1100)/Term 305 (EL2008)
//     PlcTask Inputs/GVL_iXlinker.Device_3_EtherCAT.Term_146_EK1100.Term_288_EK1122.Term_294_EK1100.Term_305_EL2008.InfoData.State <-> InfoData/State
//     PlcTask Inputs/GVL_iXlinker.Device_3_EtherCAT.Term_146_EK1100.Term_288_EK1122.Term_294_EK1100.Term_305_EL2008.WcState.WcState <-> WcState/WcState
//     PlcTask Outputs/GVL_iXlinker.Device_3_EtherCAT.Term_146_EK1100.Term_288_EK1122.Term_294_EK1100.Term_305_EL2008.Channel_{1..8}.Output <-> Channel {1..8}/Output  (8 links)
//   Plc1/Plc1 Instance <-> Device 3 (EtherCAT)/Term 146 (EK1100)/Term 288 (EK1122)/Term 307 (EK1100)
//     PlcTask Inputs/GVL_iXlinker.Device_3_EtherCAT.Term_146_EK1100.Term_288_EK1122.Term_307_EK1100.InfoData.State <-> InfoData/State
//   Plc1/Plc1 Instance <-> Device 3 (EtherCAT)/Term 146 (EK1100)/Term 288 (EK1122)/Term 307 (EK1100)/Term 330 (EK1122)
//     PlcTask Inputs/GVL_iXlinker.Device_3_EtherCAT.Term_146_EK1100.Term_288_EK1122.Term_307_EK1100.Term_330_EK1122.InfoData.State <-> InfoData/State
//   Plc1/Plc1 Instance <-> Device 3 (EtherCAT)/Term 146 (EK1100)/Term 288 (EK1122)/Term 307 (EK1100)/Term 330 (EK1122)/Term 331 (EK1100)
//     PlcTask Inputs/GVL_iXlinker.Device_3_EtherCAT.Term_146_EK1100.Term_288_EK1122.Term_307_EK1100.Term_330_EK1122.Term_331_EK1100.InfoData.State <-> InfoData/State
//   Plc1/Plc1 Instance <-> Device 3 (EtherCAT)/Term 146 (EK1100)/Term 288 (EK1122)/Term 307 (EK1100)/Term 330 (EK1122)/Term 331 (EK1100)/Term 332 (EL1809)
//     PlcTask Inputs/GVL_iXlinker.Device_3_EtherCAT.Term_146_EK1100.Term_288_EK1122.Term_307_EK1100.Term_330_EK1122.Term_331_EK1100.Term_332_EL1809.Channel_{1..16}.Input <-> Channel {1..16}/Input  (16 links)
//     PlcTask Inputs/GVL_iXlinker.Device_3_EtherCAT.Term_146_EK1100.Term_288_EK1122.Term_307_EK1100.Term_330_EK1122.Term_331_EK1100.Term_332_EL1809.InfoData.State <-> InfoData/State
//     PlcTask Inputs/GVL_iXlinker.Device_3_EtherCAT.Term_146_EK1100.Term_288_EK1122.Term_307_EK1100.Term_330_EK1122.Term_331_EK1100.Term_332_EL1809.WcState.InputToggle <-> WcState/InputToggle
//     PlcTask Inputs/GVL_iXlinker.Device_3_EtherCAT.Term_146_EK1100.Term_288_EK1122.Term_307_EK1100.Term_330_EK1122.Term_331_EK1100.Term_332_EL1809.WcState.WcState <-> WcState/WcState
//   Plc1/Plc1 Instance <-> Device 3 (EtherCAT)/Term 146 (EK1100)/Term 288 (EK1122)/Term 307 (EK1100)/Term 330 (EK1122)/Term 333 (EK1100)
//     PlcTask Inputs/GVL_iXlinker.Device_3_EtherCAT.Term_146_EK1100.Term_288_EK1122.Term_307_EK1100.Term_330_EK1122.Term_333_EK1100.InfoData.State <-> InfoData/State
//   Plc1/Plc1 Instance <-> Device 3 (EtherCAT)/Term 146 (EK1100)/Term 288 (EK1122)/Term 307 (EK1100)/Term 330 (EK1122)/Term 333 (EK1100)/Term 334 (EL1809)
//     PlcTask Inputs/GVL_iXlinker.Device_3_EtherCAT.Term_146_EK1100.Term_288_EK1122.Term_307_EK1100.Term_330_EK1122.Term_333_EK1100.Term_334_EL1809.Channel_{1..16}.Input <-> Channel {1..16}/Input  (16 links)
//     PlcTask Inputs/GVL_iXlinker.Device_3_EtherCAT.Term_146_EK1100.Term_288_EK1122.Term_307_EK1100.Term_330_EK1122.Term_333_EK1100.Term_334_EL1809.InfoData.State <-> InfoData/State
//     PlcTask Inputs/GVL_iXlinker.Device_3_EtherCAT.Term_146_EK1100.Term_288_EK1122.Term_307_EK1100.Term_330_EK1122.Term_333_EK1100.Term_334_EL1809.WcState.InputToggle <-> WcState/InputToggle
//     PlcTask Inputs/GVL_iXlinker.Device_3_EtherCAT.Term_146_EK1100.Term_288_EK1122.Term_307_EK1100.Term_330_EK1122.Term_333_EK1100.Term_334_EL1809.WcState.WcState <-> WcState/WcState
//   Plc1/Plc1 Instance <-> Device 3 (EtherCAT)/Term 146 (EK1100)/Term 288 (EK1122)/Term 307 (EK1100)/Term 335 (EL2008)
//     PlcTask Inputs/GVL_iXlinker.Device_3_EtherCAT.Term_146_EK1100.Term_288_EK1122.Term_307_EK1100.Term_335_EL2008.InfoData.State <-> InfoData/State
//     PlcTask Inputs/GVL_iXlinker.Device_3_EtherCAT.Term_146_EK1100.Term_288_EK1122.Term_307_EK1100.Term_335_EL2008.WcState.WcState <-> WcState/WcState
//     PlcTask Outputs/GVL_iXlinker.Device_3_EtherCAT.Term_146_EK1100.Term_288_EK1122.Term_307_EK1100.Term_335_EL2008.Channel_{1..8}.Output <-> Channel {1..8}/Output  (8 links)
//   Plc1/Plc1 Instance <-> Device 3 (EtherCAT)/Term 146 (EK1100)/Term 288 (EK1122)/Term 307 (EK1100)/Term 336 (EL2008)
//     PlcTask Inputs/GVL_iXlinker.Device_3_EtherCAT.Term_146_EK1100.Term_288_EK1122.Term_307_EK1100.Term_336_EL2008.InfoData.State <-> InfoData/State
//     PlcTask Inputs/GVL_iXlinker.Device_3_EtherCAT.Term_146_EK1100.Term_288_EK1122.Term_307_EK1100.Term_336_EL2008.WcState.WcState <-> WcState/WcState
//     PlcTask Outputs/GVL_iXlinker.Device_3_EtherCAT.Term_146_EK1100.Term_288_EK1122.Term_307_EK1100.Term_336_EL2008.Channel_{1..8}.Output <-> Channel {1..8}/Output  (8 links)

CONFIGURATION Plc1
    RESOURCE PLC ON TwinCAT3
        TASK PlcTask(INTERVAL := T#10ms, PRIORITY := 20);
        PROGRAM MAIN WITH PlcTask : MAIN;
    END_RESOURCE
END_CONFIGURATION

// ---- DUTs/IO/PdoEntries/Status_3D84275F.TcDUT
{attribute 'GeneratedUsingTerminal: EL6002-0000-0019'}
{attribute addProperty BoxType "EL6002-0000-0019"}
{attribute addProperty Id "Transmit_acceptedBOOL1Receive_requestBOOL1Init_acceptedBOOL1Buffer_fullBOOL1Parity_errorBOOL1Framing_errorBOOL1Overrun_errorBOOL1Input_lengthUSINT1"}
{attribute addProperty CRC "1032071007"}
{attribute addProperty Size "8"}
TYPE Status_3D84275F :
STRUCT
	{attribute addProperty Name "Transmit_accepted"}
	Transmit_accepted : BOOL;
	{attribute addProperty Name "Receive_request"}
	Receive_request : BOOL;
	{attribute addProperty Name "Init_accepted"}
	Init_accepted : BOOL;
	{attribute addProperty Name "Buffer_full"}
	Buffer_full : BOOL;
	{attribute addProperty Name "Parity_error"}
	Parity_error : BOOL;
	{attribute addProperty Name "Framing_error"}
	Framing_error : BOOL;
	{attribute addProperty Name "Overrun_error"}
	Overrun_error : BOOL;
	{attribute addProperty Name "Input_length"}
	Input_length : USINT;
END_STRUCT
END_TYPE

// ---- DUTs/IO/PdoEntries/Ctrl_1EFB4D3B.TcDUT
{attribute 'GeneratedUsingTerminal: EL6002-0000-0019'}
{attribute addProperty BoxType "EL6002-0000-0019"}
{attribute addProperty Id "Transmit_requestBOOL1Receive_acceptedBOOL1Init_requestBOOL1Send_continuousBOOL1Output_lengthUSINT1"}
{attribute addProperty CRC "519785787"}
{attribute addProperty Size "5"}
TYPE Ctrl_1EFB4D3B :
STRUCT
	{attribute addProperty Name "Transmit_request"}
	Transmit_request : BOOL;
	{attribute addProperty Name "Receive_accepted"}
	Receive_accepted : BOOL;
	{attribute addProperty Name "Init_request"}
	Init_request : BOOL;
	{attribute addProperty Name "Send_continuous"}
	Send_continuous : BOOL;
	{attribute addProperty Name "Output_length"}
	Output_length : USINT;
END_STRUCT
END_TYPE

// ---- DUTs/IO/PdoEntries/Ctrl_71604E86.TcDUT
{attribute 'GeneratedUsingTerminal: EL6001-0000-0020'}
{attribute addProperty BoxType "EL6001-0000-0020"}
{attribute addProperty Id "Transmit_requestBOOL1Receive_acceptedBOOL1Init_requestBOOL1Send_continuesBOOL1Output_lengthUSINT1"}
{attribute addProperty CRC "1902136966"}
{attribute addProperty Size "5"}
TYPE Ctrl_71604E86 :
STRUCT
	{attribute addProperty Name "Transmit_request"}
	Transmit_request : BOOL;
	{attribute addProperty Name "Receive_accepted"}
	Receive_accepted : BOOL;
	{attribute addProperty Name "Init_request"}
	Init_request : BOOL;
	{attribute addProperty Name "Send_continues"}
	Send_continues : BOOL;
	{attribute addProperty Name "Output_length"}
	Output_length : USINT;
END_STRUCT
END_TYPE

// ---- DUTs/IO/PdoEntries/Status_B0753356.TcDUT
{attribute 'GeneratedUsingTerminal: EL3174-0002-0017'}
{attribute addProperty BoxType "EL3174-0002-0017"}
{attribute addProperty Id "UnderrangeBOOL1OverrangeBOOL1Limit_1BYTE1Limit_2BYTE1ErrorBOOL1Sync_errorBOOL1TxPDO_StateBOOL1TxPDO_ToggleBOOL1"}
{attribute addProperty CRC "2960470870"}
{attribute addProperty Size "8"}
TYPE Status_B0753356 :
STRUCT
	{attribute addProperty Name "Underrange"}
	Underrange : BOOL;
	{attribute addProperty Name "Overrange"}
	Overrange : BOOL;
	{attribute addProperty Name "Limit_1"}
	Limit_1 : BYTE;
	{attribute addProperty Name "Limit_2"}
	Limit_2 : BYTE;
	{attribute addProperty Name "Error"}
	Error : BOOL;
	{attribute addProperty Name "Sync_error"}
	Sync_error : BOOL;
	{attribute addProperty Name "TxPDO_State"}
	TxPDO_State : BOOL;
	{attribute addProperty Name "TxPDO_Toggle"}
	TxPDO_Toggle : BOOL;
END_STRUCT
END_TYPE

// ---- DUTs/IO/PdoEntries/Status_F2CE6D91.TcDUT
{attribute 'GeneratedUsingTerminal: EL3011-0000-0018'}
{attribute addProperty BoxType "EL3011-0000-0018"}
{attribute addProperty Id "UnderrangeBOOL1OverrangeBOOL1Limit_1BYTE1Limit_2BYTE1ErrorBOOL1TxPDO_StateBOOL1TxPDO_ToggleBOOL1"}
{attribute addProperty CRC "4073614737"}
{attribute addProperty Size "7"}
TYPE Status_F2CE6D91 :
STRUCT
	{attribute addProperty Name "Underrange"}
	Underrange : BOOL;
	{attribute addProperty Name "Overrange"}
	Overrange : BOOL;
	{attribute addProperty Name "Limit_1"}
	Limit_1 : BYTE;
	{attribute addProperty Name "Limit_2"}
	Limit_2 : BYTE;
	{attribute addProperty Name "Error"}
	Error : BOOL;
	{attribute addProperty Name "TxPDO_State"}
	TxPDO_State : BOOL;
	{attribute addProperty Name "TxPDO_Toggle"}
	TxPDO_Toggle : BOOL;
END_STRUCT
END_TYPE

// ---- DUTs/IO/PdoEntries/U1_Status_DC903920.TcDUT
{attribute 'GeneratedUsingTerminal: EL3773-0000-0021'}
{attribute addProperty BoxType "EL3773-0000-0021"}
{attribute addProperty Id "UnderrangeBOOL1OverrangeBOOL1Limit_xBYTE1ErrorBOOL1Sync_errorBOOL1TxPDO_StateBOOL1TxPDO_ToggleBOOL1"}
{attribute addProperty CRC "3700439328"}
{attribute addProperty Size "7"}
TYPE U1_Status_DC903920 :
STRUCT
	{attribute addProperty Name "Underrange"}
	Underrange : BOOL;
	{attribute addProperty Name "Overrange"}
	Overrange : BOOL;
	{attribute addProperty Name "Limit_x"}
	Limit_x : BYTE;
	{attribute addProperty Name "Error"}
	Error : BOOL;
	{attribute addProperty Name "Sync_error"}
	Sync_error : BOOL;
	{attribute addProperty Name "TxPDO_State"}
	TxPDO_State : BOOL;
	{attribute addProperty Name "TxPDO_Toggle"}
	TxPDO_Toggle : BOOL;
END_STRUCT
END_TYPE

// ---- DUTs/IO/PdoEntries/U1_Samples_25492287.TcDUT
{attribute 'GeneratedUsingTerminal: EL3773-0000-0021'}
{attribute addProperty BoxType "EL3773-0000-0021"}
{attribute addProperty Id "ARRAY_0INT2ARRAY_1INT2ARRAY_2INT2ARRAY_3INT2ARRAY_4INT2ARRAY_5INT2ARRAY_6INT2ARRAY_7INT2ARRAY_8INT2ARRAY_9INT2"}
{attribute addProperty CRC "625549959"}
{attribute addProperty Size "20"}
TYPE U1_Samples_25492287 :
STRUCT
	{attribute addProperty Name "ARRAY_0"}
	ARRAY_0 : INT;
	{attribute addProperty Name "ARRAY_1"}
	ARRAY_1 : INT;
	{attribute addProperty Name "ARRAY_2"}
	ARRAY_2 : INT;
	{attribute addProperty Name "ARRAY_3"}
	ARRAY_3 : INT;
	{attribute addProperty Name "ARRAY_4"}
	ARRAY_4 : INT;
	{attribute addProperty Name "ARRAY_5"}
	ARRAY_5 : INT;
	{attribute addProperty Name "ARRAY_6"}
	ARRAY_6 : INT;
	{attribute addProperty Name "ARRAY_7"}
	ARRAY_7 : INT;
	{attribute addProperty Name "ARRAY_8"}
	ARRAY_8 : INT;
	{attribute addProperty Name "ARRAY_9"}
	ARRAY_9 : INT;
END_STRUCT
END_TYPE

// ---- DUTs/IO/PdoEntries/I1_Status_DC903920.TcDUT
{attribute 'GeneratedUsingTerminal: EL3773-0000-0021'}
{attribute addProperty BoxType "EL3773-0000-0021"}
{attribute addProperty Id "UnderrangeBOOL1OverrangeBOOL1Limit_xBYTE1ErrorBOOL1Sync_errorBOOL1TxPDO_StateBOOL1TxPDO_ToggleBOOL1"}
{attribute addProperty CRC "3700439328"}
{attribute addProperty Size "7"}
TYPE I1_Status_DC903920 :
STRUCT
	{attribute addProperty Name "Underrange"}
	Underrange : BOOL;
	{attribute addProperty Name "Overrange"}
	Overrange : BOOL;
	{attribute addProperty Name "Limit_x"}
	Limit_x : BYTE;
	{attribute addProperty Name "Error"}
	Error : BOOL;
	{attribute addProperty Name "Sync_error"}
	Sync_error : BOOL;
	{attribute addProperty Name "TxPDO_State"}
	TxPDO_State : BOOL;
	{attribute addProperty Name "TxPDO_Toggle"}
	TxPDO_Toggle : BOOL;
END_STRUCT
END_TYPE

// ---- DUTs/IO/PdoEntries/I1_Samples_25492287.TcDUT
{attribute 'GeneratedUsingTerminal: EL3773-0000-0021'}
{attribute addProperty BoxType "EL3773-0000-0021"}
{attribute addProperty Id "ARRAY_0INT2ARRAY_1INT2ARRAY_2INT2ARRAY_3INT2ARRAY_4INT2ARRAY_5INT2ARRAY_6INT2ARRAY_7INT2ARRAY_8INT2ARRAY_9INT2"}
{attribute addProperty CRC "625549959"}
{attribute addProperty Size "20"}
TYPE I1_Samples_25492287 :
STRUCT
	{attribute addProperty Name "ARRAY_0"}
	ARRAY_0 : INT;
	{attribute addProperty Name "ARRAY_1"}
	ARRAY_1 : INT;
	{attribute addProperty Name "ARRAY_2"}
	ARRAY_2 : INT;
	{attribute addProperty Name "ARRAY_3"}
	ARRAY_3 : INT;
	{attribute addProperty Name "ARRAY_4"}
	ARRAY_4 : INT;
	{attribute addProperty Name "ARRAY_5"}
	ARRAY_5 : INT;
	{attribute addProperty Name "ARRAY_6"}
	ARRAY_6 : INT;
	{attribute addProperty Name "ARRAY_7"}
	ARRAY_7 : INT;
	{attribute addProperty Name "ARRAY_8"}
	ARRAY_8 : INT;
	{attribute addProperty Name "ARRAY_9"}
	ARRAY_9 : INT;
END_STRUCT
END_TYPE

// ---- DUTs/IO/PdoEntries/U2_Status_DC903920.TcDUT
{attribute 'GeneratedUsingTerminal: EL3773-0000-0021'}
{attribute addProperty BoxType "EL3773-0000-0021"}
{attribute addProperty Id "UnderrangeBOOL1OverrangeBOOL1Limit_xBYTE1ErrorBOOL1Sync_errorBOOL1TxPDO_StateBOOL1TxPDO_ToggleBOOL1"}
{attribute addProperty CRC "3700439328"}
{attribute addProperty Size "7"}
TYPE U2_Status_DC903920 :
STRUCT
	{attribute addProperty Name "Underrange"}
	Underrange : BOOL;
	{attribute addProperty Name "Overrange"}
	Overrange : BOOL;
	{attribute addProperty Name "Limit_x"}
	Limit_x : BYTE;
	{attribute addProperty Name "Error"}
	Error : BOOL;
	{attribute addProperty Name "Sync_error"}
	Sync_error : BOOL;
	{attribute addProperty Name "TxPDO_State"}
	TxPDO_State : BOOL;
	{attribute addProperty Name "TxPDO_Toggle"}
	TxPDO_Toggle : BOOL;
END_STRUCT
END_TYPE

// ---- DUTs/IO/PdoEntries/U2_Samples_25492287.TcDUT
{attribute 'GeneratedUsingTerminal: EL3773-0000-0021'}
{attribute addProperty BoxType "EL3773-0000-0021"}
{attribute addProperty Id "ARRAY_0INT2ARRAY_1INT2ARRAY_2INT2ARRAY_3INT2ARRAY_4INT2ARRAY_5INT2ARRAY_6INT2ARRAY_7INT2ARRAY_8INT2ARRAY_9INT2"}
{attribute addProperty CRC "625549959"}
{attribute addProperty Size "20"}
TYPE U2_Samples_25492287 :
STRUCT
	{attribute addProperty Name "ARRAY_0"}
	ARRAY_0 : INT;
	{attribute addProperty Name "ARRAY_1"}
	ARRAY_1 : INT;
	{attribute addProperty Name "ARRAY_2"}
	ARRAY_2 : INT;
	{attribute addProperty Name "ARRAY_3"}
	ARRAY_3 : INT;
	{attribute addProperty Name "ARRAY_4"}
	ARRAY_4 : INT;
	{attribute addProperty Name "ARRAY_5"}
	ARRAY_5 : INT;
	{attribute addProperty Name "ARRAY_6"}
	ARRAY_6 : INT;
	{attribute addProperty Name "ARRAY_7"}
	ARRAY_7 : INT;
	{attribute addProperty Name "ARRAY_8"}
	ARRAY_8 : INT;
	{attribute addProperty Name "ARRAY_9"}
	ARRAY_9 : INT;
END_STRUCT
END_TYPE

// ---- DUTs/IO/PdoEntries/I2_Status_DC903920.TcDUT
{attribute 'GeneratedUsingTerminal: EL3773-0000-0021'}
{attribute addProperty BoxType "EL3773-0000-0021"}
{attribute addProperty Id "UnderrangeBOOL1OverrangeBOOL1Limit_xBYTE1ErrorBOOL1Sync_errorBOOL1TxPDO_StateBOOL1TxPDO_ToggleBOOL1"}
{attribute addProperty CRC "3700439328"}
{attribute addProperty Size "7"}
TYPE I2_Status_DC903920 :
STRUCT
	{attribute addProperty Name "Underrange"}
	Underrange : BOOL;
	{attribute addProperty Name "Overrange"}
	Overrange : BOOL;
	{attribute addProperty Name "Limit_x"}
	Limit_x : BYTE;
	{attribute addProperty Name "Error"}
	Error : BOOL;
	{attribute addProperty Name "Sync_error"}
	Sync_error : BOOL;
	{attribute addProperty Name "TxPDO_State"}
	TxPDO_State : BOOL;
	{attribute addProperty Name "TxPDO_Toggle"}
	TxPDO_Toggle : BOOL;
END_STRUCT
END_TYPE

// ---- DUTs/IO/PdoEntries/I2_Samples_25492287.TcDUT
{attribute 'GeneratedUsingTerminal: EL3773-0000-0021'}
{attribute addProperty BoxType "EL3773-0000-0021"}
{attribute addProperty Id "ARRAY_0INT2ARRAY_1INT2ARRAY_2INT2ARRAY_3INT2ARRAY_4INT2ARRAY_5INT2ARRAY_6INT2ARRAY_7INT2ARRAY_8INT2ARRAY_9INT2"}
{attribute addProperty CRC "625549959"}
{attribute addProperty Size "20"}
TYPE I2_Samples_25492287 :
STRUCT
	{attribute addProperty Name "ARRAY_0"}
	ARRAY_0 : INT;
	{attribute addProperty Name "ARRAY_1"}
	ARRAY_1 : INT;
	{attribute addProperty Name "ARRAY_2"}
	ARRAY_2 : INT;
	{attribute addProperty Name "ARRAY_3"}
	ARRAY_3 : INT;
	{attribute addProperty Name "ARRAY_4"}
	ARRAY_4 : INT;
	{attribute addProperty Name "ARRAY_5"}
	ARRAY_5 : INT;
	{attribute addProperty Name "ARRAY_6"}
	ARRAY_6 : INT;
	{attribute addProperty Name "ARRAY_7"}
	ARRAY_7 : INT;
	{attribute addProperty Name "ARRAY_8"}
	ARRAY_8 : INT;
	{attribute addProperty Name "ARRAY_9"}
	ARRAY_9 : INT;
END_STRUCT
END_TYPE

// ---- DUTs/IO/PdoEntries/U3_Status_DC903920.TcDUT
{attribute 'GeneratedUsingTerminal: EL3773-0000-0021'}
{attribute addProperty BoxType "EL3773-0000-0021"}
{attribute addProperty Id "UnderrangeBOOL1OverrangeBOOL1Limit_xBYTE1ErrorBOOL1Sync_errorBOOL1TxPDO_StateBOOL1TxPDO_ToggleBOOL1"}
{attribute addProperty CRC "3700439328"}
{attribute addProperty Size "7"}
TYPE U3_Status_DC903920 :
STRUCT
	{attribute addProperty Name "Underrange"}
	Underrange : BOOL;
	{attribute addProperty Name "Overrange"}
	Overrange : BOOL;
	{attribute addProperty Name "Limit_x"}
	Limit_x : BYTE;
	{attribute addProperty Name "Error"}
	Error : BOOL;
	{attribute addProperty Name "Sync_error"}
	Sync_error : BOOL;
	{attribute addProperty Name "TxPDO_State"}
	TxPDO_State : BOOL;
	{attribute addProperty Name "TxPDO_Toggle"}
	TxPDO_Toggle : BOOL;
END_STRUCT
END_TYPE

// ---- DUTs/IO/PdoEntries/U3_Samples_25492287.TcDUT
{attribute 'GeneratedUsingTerminal: EL3773-0000-0021'}
{attribute addProperty BoxType "EL3773-0000-0021"}
{attribute addProperty Id "ARRAY_0INT2ARRAY_1INT2ARRAY_2INT2ARRAY_3INT2ARRAY_4INT2ARRAY_5INT2ARRAY_6INT2ARRAY_7INT2ARRAY_8INT2ARRAY_9INT2"}
{attribute addProperty CRC "625549959"}
{attribute addProperty Size "20"}
TYPE U3_Samples_25492287 :
STRUCT
	{attribute addProperty Name "ARRAY_0"}
	ARRAY_0 : INT;
	{attribute addProperty Name "ARRAY_1"}
	ARRAY_1 : INT;
	{attribute addProperty Name "ARRAY_2"}
	ARRAY_2 : INT;
	{attribute addProperty Name "ARRAY_3"}
	ARRAY_3 : INT;
	{attribute addProperty Name "ARRAY_4"}
	ARRAY_4 : INT;
	{attribute addProperty Name "ARRAY_5"}
	ARRAY_5 : INT;
	{attribute addProperty Name "ARRAY_6"}
	ARRAY_6 : INT;
	{attribute addProperty Name "ARRAY_7"}
	ARRAY_7 : INT;
	{attribute addProperty Name "ARRAY_8"}
	ARRAY_8 : INT;
	{attribute addProperty Name "ARRAY_9"}
	ARRAY_9 : INT;
END_STRUCT
END_TYPE

// ---- DUTs/IO/PdoEntries/I3_Status_DC903920.TcDUT
{attribute 'GeneratedUsingTerminal: EL3773-0000-0021'}
{attribute addProperty BoxType "EL3773-0000-0021"}
{attribute addProperty Id "UnderrangeBOOL1OverrangeBOOL1Limit_xBYTE1ErrorBOOL1Sync_errorBOOL1TxPDO_StateBOOL1TxPDO_ToggleBOOL1"}
{attribute addProperty CRC "3700439328"}
{attribute addProperty Size "7"}
TYPE I3_Status_DC903920 :
STRUCT
	{attribute addProperty Name "Underrange"}
	Underrange : BOOL;
	{attribute addProperty Name "Overrange"}
	Overrange : BOOL;
	{attribute addProperty Name "Limit_x"}
	Limit_x : BYTE;
	{attribute addProperty Name "Error"}
	Error : BOOL;
	{attribute addProperty Name "Sync_error"}
	Sync_error : BOOL;
	{attribute addProperty Name "TxPDO_State"}
	TxPDO_State : BOOL;
	{attribute addProperty Name "TxPDO_Toggle"}
	TxPDO_Toggle : BOOL;
END_STRUCT
END_TYPE

// ---- DUTs/IO/PdoEntries/I3_Samples_25492287.TcDUT
{attribute 'GeneratedUsingTerminal: EL3773-0000-0021'}
{attribute addProperty BoxType "EL3773-0000-0021"}
{attribute addProperty Id "ARRAY_0INT2ARRAY_1INT2ARRAY_2INT2ARRAY_3INT2ARRAY_4INT2ARRAY_5INT2ARRAY_6INT2ARRAY_7INT2ARRAY_8INT2ARRAY_9INT2"}
{attribute addProperty CRC "625549959"}
{attribute addProperty Size "20"}
TYPE I3_Samples_25492287 :
STRUCT
	{attribute addProperty Name "ARRAY_0"}
	ARRAY_0 : INT;
	{attribute addProperty Name "ARRAY_1"}
	ARRAY_1 : INT;
	{attribute addProperty Name "ARRAY_2"}
	ARRAY_2 : INT;
	{attribute addProperty Name "ARRAY_3"}
	ARRAY_3 : INT;
	{attribute addProperty Name "ARRAY_4"}
	ARRAY_4 : INT;
	{attribute addProperty Name "ARRAY_5"}
	ARRAY_5 : INT;
	{attribute addProperty Name "ARRAY_6"}
	ARRAY_6 : INT;
	{attribute addProperty Name "ARRAY_7"}
	ARRAY_7 : INT;
	{attribute addProperty Name "ARRAY_8"}
	ARRAY_8 : INT;
	{attribute addProperty Name "ARRAY_9"}
	ARRAY_9 : INT;
END_STRUCT
END_TYPE

// ---- DUTs/IO/PdoEntries/StartTimeNextLatch_02E0C1C8.TcDUT
{attribute 'GeneratedUsingTerminal: EL3773-0000-0021'}
{attribute addProperty BoxType "EL3773-0000-0021"}
{attribute addProperty Id "LowUDINT4HiUDINT4"}
{attribute addProperty CRC "48284104"}
{attribute addProperty Size "8"}
TYPE StartTimeNextLatch_02E0C1C8 :
STRUCT
	{attribute addProperty Name "Low"}
	Low : UDINT;
	{attribute addProperty Name "Hi"}
	Hi : UDINT;
END_STRUCT
END_TYPE

// ---- DUTs/IO/PdoEntries/Status_642C2ED1.TcDUT
{attribute 'GeneratedUsingTerminal: EL2258-0000-0017'}
{attribute addProperty BoxType "EL2258-0000-0017"}
{attribute addProperty Id "Output_short_circuitBOOL1Output_buffer_overflowBOOL1Output_stateBOOL1Input_cycle_counterBYTE1Output_order_feedbackUSINT1Events_in_output_bufferUSINT1"}
{attribute addProperty CRC "1680617169"}
{attribute addProperty Size "6"}
TYPE Status_642C2ED1 :
STRUCT
	{attribute addProperty Name "Output_short_circuit"}
	Output_short_circuit : BOOL;
	{attribute addProperty Name "Output_buffer_overflow"}
	Output_buffer_overflow : BOOL;
	{attribute addProperty Name "Output_state"}
	Output_state : BOOL;
	{attribute addProperty Name "Input_cycle_counter"}
	Input_cycle_counter : BYTE;
	{attribute addProperty Name "Output_order_feedback"}
	Output_order_feedback : USINT;
	{attribute addProperty Name "Events_in_output_buffer"}
	Events_in_output_buffer : USINT;
END_STRUCT
END_TYPE

// ---- DUTs/IO/PdoEntries/Ctrl_77460BD3.TcDUT
{attribute 'GeneratedUsingTerminal: EL2258-0000-0017'}
{attribute addProperty BoxType "EL2258-0000-0017"}
{attribute addProperty Id "Output_buffer_resetBOOL1Manual_output_stateBOOL1Force_orderBOOL1Enable_manual_operationBOOL1Output_order_counterUSINT1No_of_output_eventsUSINT1"}
{attribute addProperty CRC "2001079251"}
{attribute addProperty Size "6"}
TYPE Ctrl_77460BD3 :
STRUCT
	{attribute addProperty Name "Output_buffer_reset"}
	Output_buffer_reset : BOOL;
	{attribute addProperty Name "Manual_output_state"}
	Manual_output_state : BOOL;
	{attribute addProperty Name "Force_order"}
	Force_order : BOOL;
	{attribute addProperty Name "Enable_manual_operation"}
	Enable_manual_operation : BOOL;
	{attribute addProperty Name "Output_order_counter"}
	Output_order_counter : USINT;
	{attribute addProperty Name "No_of_output_events"}
	No_of_output_events : USINT;
END_STRUCT
END_TYPE

// ---- DUTs/IO/PdoEntries/Outputs_A910484D.TcDUT
{attribute 'GeneratedUsingTerminal: EL2258-0000-0017'}
{attribute addProperty BoxType "EL2258-0000-0017"}
{attribute addProperty Id "Output_event_state_1BOOL1Output_event_state_2BOOL1Output_event_state_3BOOL1Output_event_state_4BOOL1Output_event_state_5BOOL1Output_event_state_6BOOL1Output_event_state_7BOOL1Output_event_state_8BOOL1Output_event_state_9BOOL1Output_event_state_10BOOL1"}
{attribute addProperty CRC "2836416589"}
{attribute addProperty Size "10"}
TYPE Outputs_A910484D :
STRUCT
	{attribute addProperty Name "Output_event_state_1"}
	Output_event_state_1 : BOOL;
	{attribute addProperty Name "Output_event_state_2"}
	Output_event_state_2 : BOOL;
	{attribute addProperty Name "Output_event_state_3"}
	Output_event_state_3 : BOOL;
	{attribute addProperty Name "Output_event_state_4"}
	Output_event_state_4 : BOOL;
	{attribute addProperty Name "Output_event_state_5"}
	Output_event_state_5 : BOOL;
	{attribute addProperty Name "Output_event_state_6"}
	Output_event_state_6 : BOOL;
	{attribute addProperty Name "Output_event_state_7"}
	Output_event_state_7 : BOOL;
	{attribute addProperty Name "Output_event_state_8"}
	Output_event_state_8 : BOOL;
	{attribute addProperty Name "Output_event_state_9"}
	Output_event_state_9 : BOOL;
	{attribute addProperty Name "Output_event_state_10"}
	Output_event_state_10 : BOOL;
END_STRUCT
END_TYPE

// ---- DUTs/IO/PDOs/COM_TxPDO_Map_Inputs_Channel_3801C95E.TcDUT
{attribute 'GeneratedUsingTerminal: EL6002-0000-0019'}
{attribute addProperty BoxType "EL6002-0000-0019"}
{attribute addProperty Id "StatusAT %I*Status_3D84275F8Data_InAT %I*ARRAY[0..21] OF USINT22"}
{attribute addProperty CRC "1334739266"}
{attribute addProperty Size "30"}
TYPE COM_TxPDO_Map_Inputs_Channel_3801C95E EXTENDS TcoIo.InputBase_8311D824 :
STRUCT
	{attribute addProperty Name "Status"}
	Status AT %I* : Status_3D84275F;
	{attribute addProperty Name "Data_In"}
	Data_In AT %I* : ARRAY[0..21] OF USINT;
END_STRUCT
END_TYPE

// ---- DUTs/IO/PDOs/COM_RxPDO_Map_Outputs_Channel_EADA2E0D.TcDUT
{attribute 'GeneratedUsingTerminal: EL6002-0000-0019'}
{attribute addProperty BoxType "EL6002-0000-0019"}
{attribute addProperty Id "CtrlAT %Q*Ctrl_1EFB4D3B5Data_OutAT %Q*ARRAY[0..21] OF USINT22"}
{attribute addProperty CRC "3494673196"}
{attribute addProperty Size "27"}
TYPE COM_RxPDO_Map_Outputs_Channel_EADA2E0D EXTENDS TcoIo.OutputBase_10CEE7DE :
STRUCT
	{attribute addProperty Name "Ctrl"}
	Ctrl AT %Q* : Ctrl_1EFB4D3B;
	{attribute addProperty Name "Data_Out"}
	Data_Out AT %Q* : ARRAY[0..21] OF USINT;
END_STRUCT
END_TYPE

// ---- DUTs/IO/PDOs/Channel_830843C1.TcDUT
{attribute 'GeneratedUsingTerminal: EL1809-0000-0018'}
{attribute addProperty BoxType "EL1809-0000-0018"}
{attribute addProperty Id "InputAT %I*BOOL1"}
{attribute addProperty CRC "2198356929"}
{attribute addProperty Size "1"}
TYPE Channel_830843C1 EXTENDS TcoIo.InputBase_8311D824 :
STRUCT
	{attribute addProperty Name "Input"}
	Input AT %I* : BOOL;
END_STRUCT
END_TYPE

// ---- DUTs/IO/PDOs/Channel_42CA91F7.TcDUT
{attribute 'GeneratedUsingTerminal: EL2809-0000-0018'}
{attribute addProperty BoxType "EL2809-0000-0018"}
{attribute addProperty Id "OutputAT %Q*BOOL1"}
{attribute addProperty CRC "1120571895"}
{attribute addProperty Size "1"}
TYPE Channel_42CA91F7 EXTENDS TcoIo.OutputBase_10CEE7DE :
STRUCT
	{attribute addProperty Name "Output"}
	Output AT %Q* : BOOL;
END_STRUCT
END_TYPE

// ---- DUTs/IO/PDOs/AO_Output_Channel_BA7EBB7C.TcDUT
{attribute 'GeneratedUsingTerminal: EL4004-0000-0020'}
{attribute addProperty BoxType "EL4004-0000-0020"}
{attribute addProperty Id "Analog_outputAT %Q*INT2"}
{attribute addProperty CRC "3128867708"}
{attribute addProperty Size "2"}
TYPE AO_Output_Channel_BA7EBB7C EXTENDS TcoIo.OutputBase_10CEE7DE :
STRUCT
	{attribute addProperty Name "Analog_output"}
	Analog_output AT %Q* : INT;
END_STRUCT
END_TYPE

// ---- DUTs/IO/PDOs/COM_Inputs_3801C95E.TcDUT
{attribute 'GeneratedUsingTerminal: EL6001-0000-0020'}
{attribute addProperty BoxType "EL6001-0000-0020"}
{attribute addProperty Id "StatusAT %I*Status_3D84275F8Data_InAT %I*ARRAY[0..21] OF USINT22"}
{attribute addProperty CRC "1334739266"}
{attribute addProperty Size "30"}
TYPE COM_Inputs_3801C95E EXTENDS TcoIo.InputBase_8311D824 :
STRUCT
	{attribute addProperty Name "Status"}
	Status AT %I* : Status_3D84275F;
	{attribute addProperty Name "Data_In"}
	Data_In AT %I* : ARRAY[0..21] OF USINT;
END_STRUCT
END_TYPE

// ---- DUTs/IO/PDOs/COM_Outputs_DEF408EC.TcDUT
{attribute 'GeneratedUsingTerminal: EL6001-0000-0020'}
{attribute addProperty BoxType "EL6001-0000-0020"}
{attribute addProperty Id "CtrlAT %Q*Ctrl_71604E865Data_OutAT %Q*ARRAY[0..21] OF USINT22"}
{attribute addProperty CRC "2695605661"}
{attribute addProperty Size "27"}
TYPE COM_Outputs_DEF408EC EXTENDS TcoIo.OutputBase_10CEE7DE :
STRUCT
	{attribute addProperty Name "Ctrl"}
	Ctrl AT %Q* : Ctrl_71604E86;
	{attribute addProperty Name "Data_Out"}
	Data_Out AT %Q* : ARRAY[0..21] OF USINT;
END_STRUCT
END_TYPE

// ---- DUTs/IO/PDOs/AI_Standard_Channel_A8DF64E3.TcDUT
{attribute 'GeneratedUsingTerminal: EL3174-0002-0017'}
{attribute addProperty BoxType "EL3174-0002-0017"}
{attribute addProperty Id "StatusAT %I*Status_B07533568ValueAT %I*INT2"}
{attribute addProperty CRC "2833212643"}
{attribute addProperty Size "10"}
TYPE AI_Standard_Channel_A8DF64E3 EXTENDS TcoIo.InputBase_8311D824 :
STRUCT
	{attribute addProperty Name "Status"}
	Status AT %I* : Status_B0753356;
	{attribute addProperty Name "Value"}
	Value AT %I* : INT;
END_STRUCT
END_TYPE

// ---- DUTs/IO/PDOs/AI_Standard_Channel_4A394481.TcDUT
{attribute 'GeneratedUsingTerminal: EL3011-0000-0018'}
{attribute addProperty BoxType "EL3011-0000-0018"}
{attribute addProperty Id "StatusAT %I*Status_F2CE6D917ValueAT %I*INT2"}
{attribute addProperty CRC "1245267073"}
{attribute addProperty Size "9"}
TYPE AI_Standard_Channel_4A394481 EXTENDS TcoIo.InputBase_8311D824 :
STRUCT
	{attribute addProperty Name "Status"}
	Status AT %I* : Status_F2CE6D91;
	{attribute addProperty Name "Value"}
	Value AT %I* : INT;
END_STRUCT
END_TYPE

// ---- DUTs/IO/PDOs/L1_Voltage_Status_7371B043.TcDUT
{attribute 'GeneratedUsingTerminal: EL3773-0000-0021'}
{attribute addProperty BoxType "EL3773-0000-0021"}
{attribute addProperty Id "U1_StatusAT %I*U1_Status_DC9039207"}
{attribute addProperty CRC "1936830531"}
{attribute addProperty Size "7"}
TYPE L1_Voltage_Status_7371B043 EXTENDS TcoIo.InputBase_8311D824 :
STRUCT
	{attribute addProperty Name "U1_Status"}
	U1_Status AT %I* : U1_Status_DC903920;
END_STRUCT
END_TYPE

// ---- DUTs/IO/PDOs/L1_Voltage_Samples_41AEB7FF.TcDUT
{attribute 'GeneratedUsingTerminal: EL3773-0000-0021'}
{attribute addProperty BoxType "EL3773-0000-0021"}
{attribute addProperty Id "U1_SamplesAT %I*U1_Samples_2549228720"}
{attribute addProperty CRC "1101969407"}
{attribute addProperty Size "20"}
TYPE L1_Voltage_Samples_41AEB7FF EXTENDS TcoIo.InputBase_8311D824 :
STRUCT
	{attribute addProperty Name "U1_Samples"}
	U1_Samples AT %I* : U1_Samples_25492287;
END_STRUCT
END_TYPE

